      "I492.7" { ExternalVisible := 'False'} : Bool := FALSE;   // I492.7
      "I493.0" { ExternalVisible := 'False'} : Bool := FALSE;   // I493.0
      "I493.1" { ExternalVisible := 'False'} : Bool := FALSE;   // I493.1
      "I493.2" { ExternalVisible := 'False'} : Bool := FALSE;   // I493.2
      "I493.3" { ExternalVisible := 'False'} : Bool := FALSE;   // I493.3
      "I493.4" { ExternalVisible := 'False'} : Bool := FALSE;   // I493.4
      "I493.5" { ExternalVisible := 'False'} : Bool := FALSE;   // I493.5
      "I493.6" { ExternalVisible := 'False'} : Bool := FALSE;   // I493.6
      "I493.7" { ExternalVisible := 'False'} : Bool := FALSE;   // I493.7
      "I494.0" { ExternalVisible := 'False'} : Bool := FALSE;   // I494.0
      "I494.1" { ExternalVisible := 'False'} : Bool := FALSE;   // I494.1
      "I494.2" { ExternalVisible := 'False'} : Bool := FALSE;   // I494.2
      "I494.3" { ExternalVisible := 'False'} : Bool := FALSE;   // I494.3
      "I494.4" { ExternalVisible := 'False'} : Bool := FALSE;   // I494.4
      "I494.5" { ExternalVisible := 'False'} : Bool := FALSE;   // I494.5
      "I494.6" { ExternalVisible := 'False'} : Bool := FALSE;   // I494.6
      "I494.7" { ExternalVisible := 'False'} : Bool := FALSE;   // I494.7
      "I495.0" { ExternalVisible := 'False'} : Bool := FALSE;   // I495.0
      "I495.1" { ExternalVisible := 'False'} : Bool := FALSE;   // I495.1
      "I495.2" { ExternalVisible := 'False'} : Bool := FALSE;   // I495.2
      "I495.3" { ExternalVisible := 'False'} : Bool := FALSE;   // I495.3
      "I495.4" { ExternalVisible := 'False'} : Bool := FALSE;   // I495.4
      "I495.5" { ExternalVisible := 'False'} : Bool := FALSE;   // I495.5
      "I495.6" { ExternalVisible := 'False'} : Bool := FALSE;   // I495.6
      "I495.7" { ExternalVisible := 'False'} : Bool := FALSE;   // I495.7
      "I496.0" { ExternalVisible := 'False'} : Bool := FALSE;   // I496.0
      "I496.1" { ExternalVisible := 'False'} : Bool := FALSE;   // I496.1
      "I496.2" { ExternalVisible := 'False'} : Bool := FALSE;   // I496.2
      "I496.3" { ExternalVisible := 'False'} : Bool := FALSE;   // I496.3
      "I496.4" { ExternalVisible := 'False'} : Bool := FALSE;   // I496.4
      "I496.5" { ExternalVisible := 'False'} : Bool := FALSE;   // I496.5
      "I496.6" { ExternalVisible := 'False'} : Bool := FALSE;   // I496.6
      "I496.7" { ExternalVisible := 'False'} : Bool := FALSE;   // I496.7
      "I497.0" { ExternalVisible := 'False'} : Bool := FALSE;   // I497.0
      "I497.1" { ExternalVisible := 'False'} : Bool := FALSE;   // I497.1
      "I497.2" { ExternalVisible := 'False'} : Bool := FALSE;   // I497.2
      "I497.3" { ExternalVisible := 'False'} : Bool := FALSE;   // I497.3
      "I497.4" { ExternalVisible := 'False'} : Bool := FALSE;   // I497.4
      "I497.5" { ExternalVisible := 'False'} : Bool := FALSE;   // I497.5
      "I497.6" { ExternalVisible := 'False'} : Bool := FALSE;   // I497.6
      "I497.7" { ExternalVisible := 'False'} : Bool := FALSE;   // I497.7
      "I498.0" { ExternalVisible := 'False'} : Bool := FALSE;   // I498.0
      "I498.1" { ExternalVisible := 'False'} : Bool := FALSE;   // I498.1
      "I498.2" { ExternalVisible := 'False'} : Bool := FALSE;   // I498.2
      "I498.3" { ExternalVisible := 'False'} : Bool := FALSE;   // I498.3
      "I498.4" { ExternalVisible := 'False'} : Bool := FALSE;   // I498.4
      "I498.5" { ExternalVisible := 'False'} : Bool := FALSE;   // I498.5
      "I498.6" { ExternalVisible := 'False'} : Bool := FALSE;   // I498.6
      "I498.7" { ExternalVisible := 'False'} : Bool := FALSE;   // I498.7
      "I499.0" { ExternalVisible := 'False'} : Bool := FALSE;   // I499.0
      "I499.1" { ExternalVisible := 'False'} : Bool := FALSE;   // I499.1
      "I499.2" { ExternalVisible := 'False'} : Bool := FALSE;   // I499.2
      "I499.3" { ExternalVisible := 'False'} : Bool := FALSE;   // I499.3
      "I499.4" { ExternalVisible := 'False'} : Bool := FALSE;   // I499.4
      "I499.5" { ExternalVisible := 'False'} : Bool := FALSE;   // I499.5
      "I499.6" { ExternalVisible := 'False'} : Bool := FALSE;   // I499.6
      "I499.7" { ExternalVisible := 'False'} : Bool := FALSE;   // I499.7
      V01_Home { ExternalVisible := 'False'} : Bool := FALSE;   // 送料气缸缩回
      "V01-Work" { ExternalVisible := 'False'} : Bool := FALSE;   // 送料气缸伸出
      "V02-Home" { ExternalVisible := 'False'} : Bool := FALSE;   // 定子定位气缸缩回
      "V02-Work" { ExternalVisible := 'False'} : Bool := FALSE;   // 定子定位气缸伸出
      "V03-Home" { ExternalVisible := 'False'} : Bool := FALSE;   // 压紧气缸缩回
      "V03-Work" { ExternalVisible := 'False'} : Bool := FALSE;   // 压紧气缸伸出
      "V04-Home1" { ExternalVisible := 'False'} : Bool := FALSE;   // 纸切断气缸1缩回
      "V04-Work1" { ExternalVisible := 'False'} : Bool := FALSE;   // 纸切断气缸1伸出
      V05_Home1 { ExternalVisible := 'False'} : Bool := FALSE;   // 产品推出气缸1缩回
      V05_Work1 { ExternalVisible := 'False'} : Bool := FALSE;   // 产品推出气缸1伸出
      V06_Home1 { ExternalVisible := 'False'} : Bool := FALSE;   // 推纸气缸1缩回
      V06_Work1 { ExternalVisible := 'False'} : Bool := FALSE;   // 推纸气缸1伸出
      V07_Home1 { ExternalVisible := 'False'} : Bool := FALSE;   // 纸夹持气缸1缩回
      V07_Work1 { ExternalVisible := 'False'} : Bool := FALSE;   // 纸夹持气缸1伸出
      V08_Home1 { ExternalVisible := 'False'} : Bool := FALSE;   // 压纸气缸1缩回
      V08_Work1 { ExternalVisible := 'False'} : Bool := FALSE;   // 压纸气缸1伸出
      PX1 { ExternalVisible := 'False'} : Bool := FALSE;   // 左侧绝缘纸插入到位传感器
      PX2 { ExternalVisible := 'False'} : Bool := FALSE;   // 右侧绝缘纸插入到位传感器
      PX3 { ExternalVisible := 'False'} : Bool := FALSE;   // 左侧纸有无检测传感器
      PX4 { ExternalVisible := 'False'} : Bool := FALSE;   // 右侧纸有无检测传感器
      PX5 { ExternalVisible := 'False'} : Bool := FALSE;   // 左侧纸长限位1
      PX6 { ExternalVisible := 'False'} : Bool := FALSE;   // 左侧纸长限位2
      "V04-Home2" { ExternalVisible := 'False'} : Bool := FALSE;   // 纸切断气缸2缩回
      "V04-Work2" { ExternalVisible := 'False'} : Bool := FALSE;   // 纸切断气缸2伸出
      V05_Home2 { ExternalVisible := 'False'} : Bool := FALSE;   // 产品推出气缸2缩回
      V05_Work2 { ExternalVisible := 'False'} : Bool := FALSE;   // 产品推出气缸2伸出
      V06_Home2 { ExternalVisible := 'False'} : Bool := FALSE;   // 推纸气缸2缩回
      V06_Work2 { ExternalVisible := 'False'} : Bool := FALSE;   // 推纸气缸2伸出
      V07_Home2 { ExternalVisible := 'False'} : Bool := FALSE;   // 纸夹持气缸2缩回
      V07_Work2 { ExternalVisible := 'False'} : Bool := FALSE;   // 纸夹持气缸伸出
      V08_Home2 { ExternalVisible := 'False'} : Bool := FALSE;   // 压纸气缸2缩回
      V08_Work2 { ExternalVisible := 'False'} : Bool := FALSE;   // 压纸气缸2伸出
      V09_Home { ExternalVisible := 'False'} : Bool := FALSE;   // 定位开关气缸缩回
      "V09-Work" { ExternalVisible := 'False'} : Bool := FALSE;   // 定位开关气缸伸出
      PX7 { ExternalVisible := 'False'} : Bool := FALSE;   // 右侧纸长限位1
      PX8 { ExternalVisible := 'False'} : Bool := FALSE;   // 右侧纸长限位2
      "I504.4" { ExternalVisible := 'False'} : Bool := FALSE;   // 备用
      "I504.5" { ExternalVisible := 'False'} : Bool := FALSE;   // 备用
      "I504.6" { ExternalVisible := 'False'} : Bool := FALSE;   // 备用
      "I504.7" { ExternalVisible := 'False'} : Bool := FALSE;   // 备用
      "I505.0" { ExternalVisible := 'False'} : Bool := FALSE;   // 备用
      "I505.1" { ExternalVisible := 'False'} : Bool := FALSE;   // 备用
      "I505.2" { ExternalVisible := 'False'} : Bool := FALSE;   // 备用
      "I505.3" { ExternalVisible := 'False'} : Bool := FALSE;   // 备用
      "I505.4" { ExternalVisible := 'False'} : Bool := FALSE;   // 备用
      "I505.5" { ExternalVisible := 'False'} : Bool := FALSE;   // 备用
      "I505.6" { ExternalVisible := 'False'} : Bool := FALSE;   // 备用
      "I505.7" { ExternalVisible := 'False'} : Bool := FALSE;   // 备用
      "I506.0" { ExternalVisible := 'False'} : Bool := FALSE;   // I506.0
      "I506.1" { ExternalVisible := 'False'} : Bool := FALSE;   // I506.1
      "I506.2" { ExternalVisible := 'False'} : Bool := FALSE;   // I506.2
      "I506.3" { ExternalVisible := 'False'} : Bool := FALSE;   // I506.3
      "I506.4" { ExternalVisible := 'False'} : Bool := FALSE;   // I506.4
      "I506.5" { ExternalVisible := 'False'} : Bool := FALSE;   // I506.5
      "I506.6" { ExternalVisible := 'False'} : Bool := FALSE;   // I506.6
      "I506.7" { ExternalVisible := 'False'} : Bool := FALSE;   // I506.7
      "I507.0" { ExternalVisible := 'False'} : Bool := FALSE;   // I507.0
      "I507.1" { ExternalVisible := 'False'} : Bool := FALSE;   // I507.1
      "I507.2" { ExternalVisible := 'False'} : Bool := FALSE;   // I507.2
      "I507.3" { ExternalVisible := 'False'} : Bool := FALSE;   // I507.3
      "I507.4" { ExternalVisible := 'False'} : Bool := FALSE;   // I507.4
      "I507.5" { ExternalVisible := 'False'} : Bool := FALSE;   // I507.5
      "I507.6" { ExternalVisible := 'False'} : Bool := FALSE;   // I507.6
      "I507.7" { ExternalVisible := 'False'} : Bool := FALSE;   // I507.7
      "I508.0" { ExternalVisible := 'False'} : Bool := FALSE;   // I508.0
      "I508.1" { ExternalVisible := 'False'} : Bool := FALSE;   // I508.1
      "I508.2" { ExternalVisible := 'False'} : Bool := FALSE;   // I508.2
      "I508.3" { ExternalVisible := 'False'} : Bool := FALSE;   // I508.3
      "I508.4" { ExternalVisible := 'False'} : Bool := FALSE;   // I508.4
      "I508.5" { ExternalVisible := 'False'} : Bool := FALSE;   // I508.5
      "I508.6" { ExternalVisible := 'False'} : Bool := FALSE;   // I508.6
      "I508.7" { ExternalVisible := 'False'} : Bool := FALSE;   // I508.7
      "I509.0" { ExternalVisible := 'False'} : Bool := FALSE;   // I509.0
      "I509.1" { ExternalVisible := 'False'} : Bool := FALSE;   // I509.1
      "I509.2" { ExternalVisible := 'False'} : Bool := FALSE;   // I509.2
      "I509.3" { ExternalVisible := 'False'} : Bool := FALSE;   // I509.3
      "I509.4" { ExternalVisible := 'False'} : Bool := FALSE;   // I509.4
      "I509.5" { ExternalVisible := 'False'} : Bool := FALSE;   // I509.5
      "I509.6" { ExternalVisible := 'False'} : Bool := FALSE;   // I509.6
      "I509.7" { ExternalVisible := 'False'} : Bool := FALSE;   // I509.7
      "I510.0" { ExternalVisible := 'False'} : Bool := FALSE;   // I510.0
      "I510.1" { ExternalVisible := 'False'} : Bool := FALSE;   // I510.1
      "I510.2" { ExternalVisible := 'False'} : Bool := FALSE;   // I510.2
      "I510.3" { ExternalVisible := 'False'} : Bool := FALSE;   // I510.3
      "I510.4" { ExternalVisible := 'False'} : Bool := FALSE;   // I510.4
      "I510.5" { ExternalVisible := 'False'} : Bool := FALSE;   // I510.5
      "I510.6" { ExternalVisible := 'False'} : Bool := FALSE;   // I510.6
      "I510.7" { ExternalVisible := 'False'} : Bool := FALSE;   // I510.7
      "I511.0" { ExternalVisible := 'False'} : Bool := FALSE;   // I511.0
      "I511.1" { ExternalVisible := 'False'} : Bool := FALSE;   // I511.1
      "I511.2" { ExternalVisible := 'False'} : Bool := FALSE;   // I511.2
      "I511.3" { ExternalVisible := 'False'} : Bool := FALSE;   // I511.3
      "I511.4" { ExternalVisible := 'False'} : Bool := FALSE;   // I511.4
      "I511.5" { ExternalVisible := 'False'} : Bool := FALSE;   // I511.5
      "I511.6" { ExternalVisible := 'False'} : Bool := FALSE;   // I511.6
      "I511.7" { ExternalVisible := 'False'} : Bool := FALSE;   // I511.7
      "I512.0" { ExternalVisible := 'False'} : Bool := FALSE;   // I512.0
      "I512.1" { ExternalVisible := 'False'} : Bool := FALSE;   // I512.1
      "I512.2" { ExternalVisible := 'False'} : Bool := FALSE;   // I512.2
      "I512.3" { ExternalVisible := 'False'} : Bool := FALSE;   // I512.3
      "I512.4" { ExternalVisible := 'False'} : Bool := FALSE;   // I512.4
      "I512.5" { ExternalVisible := 'False'} : Bool := FALSE;   // I512.5
      "I512.6" { ExternalVisible := 'False'} : Bool := FALSE;   // I512.6
      "I512.7" { ExternalVisible := 'False'} : Bool := FALSE;   // I512.7
      "I513.0" { ExternalVisible := 'False'} : Bool := FALSE;   // I513.0
      "I513.1" { ExternalVisible := 'False'} : Bool := FALSE;   // I513.1
      "I513.2" { ExternalVisible := 'False'} : Bool := FALSE;   // I513.2
      "I513.3" { ExternalVisible := 'False'} : Bool := FALSE;   // I513.3
      "I513.4" { ExternalVisible := 'False'} : Bool := FALSE;   // I513.4
      "I513.5" { ExternalVisible := 'False'} : Bool := FALSE;   // I513.5
      "I513.6" { ExternalVisible := 'False'} : Bool := FALSE;   // I513.6
      "I513.7" { ExternalVisible := 'False'} : Bool := FALSE;   // I513.7
      "I514.0" { ExternalVisible := 'False'} : Bool := FALSE;   // I514.0
      "I514.1" { ExternalVisible := 'False'} : Bool := FALSE;   // I514.1
      "I514.2" { ExternalVisible := 'False'} : Bool := FALSE;   // I514.2
      "I514.3" { ExternalVisible := 'False'} : Bool := FALSE;   // I514.3
      "I514.4" { ExternalVisible := 'False'} : Bool := FALSE;   // I514.4
      "I514.5" { ExternalVisible := 'False'} : Bool := FALSE;   // I514.5
      "I514.6" { ExternalVisible := 'False'} : Bool := FALSE;   // I514.6
      "I514.7" { ExternalVisible := 'False'} : Bool := FALSE;   // I514.7
      "I515.0" { ExternalVisible := 'False'} : Bool := FALSE;   // I515.0
      "I515.1" { ExternalVisible := 'False'} : Bool := FALSE;   // I515.1
      "I515.2" { ExternalVisible := 'False'} : Bool := FALSE;   // I515.2
      "I515.3" { ExternalVisible := 'False'} : Bool := FALSE;   // I515.3
      "I515.4" { ExternalVisible := 'False'} : Bool := FALSE;   // I515.4
      "I515.5" { ExternalVisible := 'False'} : Bool := FALSE;   // I515.5
      "I515.6" { ExternalVisible := 'False'} : Bool := FALSE;   // I515.6
      "I515.7" { ExternalVisible := 'False'} : Bool := FALSE;   // I515.7
      "I516.0" { ExternalVisible := 'False'} : Bool := FALSE;   // I516.0
      "I516.1" { ExternalVisible := 'False'} : Bool := FALSE;   // I516.1
      "I516.2" { ExternalVisible := 'False'} : Bool := FALSE;   // I516.2
      "I516.3" { ExternalVisible := 'False'} : Bool := FALSE;   // I516.3
      "I516.4" { ExternalVisible := 'False'} : Bool := FALSE;   // I516.4
      "I516.5" { ExternalVisible := 'False'} : Bool := FALSE;   // I516.5
      "I516.6" { ExternalVisible := 'False'} : Bool := FALSE;   // I516.6
      "I516.7" { ExternalVisible := 'False'} : Bool := FALSE;   // I516.7
      "I517.0" { ExternalVisible := 'False'} : Bool := FALSE;   // I517.0
      "I517.1" { ExternalVisible := 'False'} : Bool := FALSE;   // I517.1
      "I517.2" { ExternalVisible := 'False'} : Bool := FALSE;   // I517.2
      "I517.3" { ExternalVisible := 'False'} : Bool := FALSE;   // I517.3
      "I517.4" { ExternalVisible := 'False'} : Bool := FALSE;   // I517.4
      "I517.5" { ExternalVisible := 'False'} : Bool := FALSE;   // I517.5
      "I517.6" { ExternalVisible := 'False'} : Bool := FALSE;   // I517.6
      "I517.7" { ExternalVisible := 'False'} : Bool := FALSE;   // I517.7
      "I518.0" { ExternalVisible := 'False'} : Bool := FALSE;   // I518.0
      "I518.1" { ExternalVisible := 'False'} : Bool := FALSE;   // I518.1
      "I518.2" { ExternalVisible := 'False'} : Bool := FALSE;   // I518.2
      "I518.3" { ExternalVisible := 'False'} : Bool := FALSE;   // I518.3
      "I518.4" { ExternalVisible := 'False'} : Bool := FALSE;   // I518.4
      "I518.5" { ExternalVisible := 'False'} : Bool := FALSE;   // I518.5
      "I518.6" { ExternalVisible := 'False'} : Bool := FALSE;   // I518.6
      "I518.7" { ExternalVisible := 'False'} : Bool := FALSE;   // I518.7
      "I519.0" { ExternalVisible := 'False'} : Bool := FALSE;   // I519.0
      "I519.1" { ExternalVisible := 'False'} : Bool := FALSE;   // I519.1
      "I519.2" { ExternalVisible := 'False'} : Bool := FALSE;   // I519.2
      "I519.3" { ExternalVisible := 'False'} : Bool := FALSE;   // I519.3
      "I519.4" { ExternalVisible := 'False'} : Bool := FALSE;   // I519.4
      "I519.5" { ExternalVisible := 'False'} : Bool := FALSE;   // I519.5
      "I519.6" { ExternalVisible := 'False'} : Bool := FALSE;   // I519.6
      "I519.7" { ExternalVisible := 'False'} : Bool := FALSE;   // I519.7
      "I520.0" { ExternalVisible := 'False'} : Bool := FALSE;   // I520.0
      "I520.1" { ExternalVisible := 'False'} : Bool := FALSE;   // I520.1
      "I520.2" { ExternalVisible := 'False'} : Bool := FALSE;   // I520.2
      "I520.3" { ExternalVisible := 'False'} : Bool := FALSE;   // I520.3
      "I520.4" { ExternalVisible := 'False'} : Bool := FALSE;   // I520.4
      "I520.5" { ExternalVisible := 'False'} : Bool := FALSE;   // I520.5
      "I520.6" { ExternalVisible := 'False'} : Bool := FALSE;   // I520.6
      "I520.7" { ExternalVisible := 'False'} : Bool := FALSE;   // I520.7
      "I521.0" { ExternalVisible := 'False'} : Bool := FALSE;   // I521.0
      "I521.1" { ExternalVisible := 'False'} : Bool := FALSE;   // I521.1
      "I521.2" { ExternalVisible := 'False'} : Bool := FALSE;   // I521.2
      "I521.3" { ExternalVisible := 'False'} : Bool := FALSE;   // I521.3
      "I521.4" { ExternalVisible := 'False'} : Bool := FALSE;   // I521.4
      "I521.5" { ExternalVisible := 'False'} : Bool := FALSE;   // I521.5
      "I521.6" { ExternalVisible := 'False'} : Bool := FALSE;   // I521.6
      "I521.7" { ExternalVisible := 'False'} : Bool := FALSE;   // I521.7
      "I522.0" { ExternalVisible := 'False'} : Bool := FALSE;   // I522.0
      "I522.1" { ExternalVisible := 'False'} : Bool := FALSE;   // I522.1
      "I522.2" { ExternalVisible := 'False'} : Bool := FALSE;   // I522.2
      "I522.3" { ExternalVisible := 'False'} : Bool := FALSE;   // I522.3
      "I522.4" { ExternalVisible := 'False'} : Bool := FALSE;   // I522.4
      "I522.5" { ExternalVisible := 'False'} : Bool := FALSE;   // I522.5
      "I522.6" { ExternalVisible := 'False'} : Bool := FALSE;   // I522.6
      "I522.7" { ExternalVisible := 'False'} : Bool := FALSE;   // I522.7
      "I523.0" { ExternalVisible := 'False'} : Bool := FALSE;   // I523.0
      "I523.1" { ExternalVisible := 'False'} : Bool := FALSE;   // I523.1
      "I523.2" { ExternalVisible := 'False'} : Bool := FALSE;   // I523.2
      "I523.3" { ExternalVisible := 'False'} : Bool := FALSE;   // I523.3
      "I523.4" { ExternalVisible := 'False'} : Bool := FALSE;   // I523.4
      "I523.5" { ExternalVisible := 'False'} : Bool := FALSE;   // I523.5
      "I523.6" { ExternalVisible := 'False'} : Bool := FALSE;   // I523.6
      "I523.7" { ExternalVisible := 'False'} : Bool := FALSE;   // I523.7
      "I524.0" { ExternalVisible := 'False'} : Bool := FALSE;   // I524.0
      "I524.1" { ExternalVisible := 'False'} : Bool := FALSE;   // I524.1
      "I524.2" { ExternalVisible := 'False'} : Bool := FALSE;   // I524.2
      "I524.3" { ExternalVisible := 'False'} : Bool := FALSE;   // I524.3
      "I524.4" { ExternalVisible := 'False'} : Bool := FALSE;   // I524.4
      "I524.5" { ExternalVisible := 'False'} : Bool := FALSE;   // I524.5
      "I524.6" { ExternalVisible := 'False'} : Bool := FALSE;   // I524.6
      "I524.7" { ExternalVisible := 'False'} : Bool := FALSE;   // I524.7
      "I525.0" { ExternalVisible := 'False'} : Bool := FALSE;   // I525.0
      "I525.1" { ExternalVisible := 'False'} : Bool := FALSE;   // I525.1
      "I525.2" { ExternalVisible := 'False'} : Bool := FALSE;   // I525.2
      "I525.3" { ExternalVisible := 'False'} : Bool := FALSE;   // I525.3
      "I525.4" { ExternalVisible := 'False'} : Bool := FALSE;   // I525.4
      "I525.5" { ExternalVisible := 'False'} : Bool := FALSE;   // I525.5
      "I525.6" { ExternalVisible := 'False'} : Bool := FALSE;   // I525.6
      "I525.7" { ExternalVisible := 'False'} : Bool := FALSE;   // I525.7
      "I526.0" { ExternalVisible := 'False'} : Bool := FALSE;   // I526.0
      "I526.1" { ExternalVisible := 'False'} : Bool := FALSE;   // I526.1
      "I526.2" { ExternalVisible := 'False'} : Bool := FALSE;   // I526.2
      "I526.3" { ExternalVisible := 'False'} : Bool := FALSE;   // I526.3
      "I526.4" { ExternalVisible := 'False'} : Bool := FALSE;   // I526.4
      "I526.5" { ExternalVisible := 'False'} : Bool := FALSE;   // I526.5
      "I526.6" { ExternalVisible := 'False'} : Bool := FALSE;   // I526.6
      "I526.7" { ExternalVisible := 'False'} : Bool := FALSE;   // I526.7
      "I527.0" { ExternalVisible := 'False'} : Bool := FALSE;   // I527.0
      "I527.1" { ExternalVisible := 'False'} : Bool := FALSE;   // I527.1
      "I527.2" { ExternalVisible := 'False'} : Bool := FALSE;   // I527.2
      "I527.3" { ExternalVisible := 'False'} : Bool := FALSE;   // I527.3
      "I527.4" { ExternalVisible := 'False'} : Bool := FALSE;   // I527.4
      "I527.5" { ExternalVisible := 'False'} : Bool := FALSE;   // I527.5
      "I527.6" { ExternalVisible := 'False'} : Bool := FALSE;   // I527.6
      "I527.7" { ExternalVisible := 'False'} : Bool := FALSE;   // I527.7
      "I528.0" { ExternalVisible := 'False'} : Bool := FALSE;   // I528.0
      "I528.1" { ExternalVisible := 'False'} : Bool := FALSE;   // I528.1
      "I528.2" { ExternalVisible := 'False'} : Bool := FALSE;   // I528.2
      "I528.3" { ExternalVisible := 'False'} : Bool := FALSE;   // I528.3
      "I528.4" { ExternalVisible := 'False'} : Bool := FALSE;   // I528.4
      "I528.5" { ExternalVisible := 'False'} : Bool := FALSE;   // I528.5
      "I528.6" { ExternalVisible := 'False'} : Bool := FALSE;   // I528.6
      "I528.7" { ExternalVisible := 'False'} : Bool := FALSE;   // I528.7
      "I529.0" { ExternalVisible := 'False'} : Bool := FALSE;   // I529.0
      "I529.1" { ExternalVisible := 'False'} : Bool := FALSE;   // I529.1
      "I529.2" { ExternalVisible := 'False'} : Bool := FALSE;   // I529.2
      "I529.3" { ExternalVisible := 'False'} : Bool := FALSE;   // I529.3
      "I529.4" { ExternalVisible := 'False'} : Bool := FALSE;   // I529.4
      "I529.5" { ExternalVisible := 'False'} : Bool := FALSE;   // I529.5
      "I529.6" { ExternalVisible := 'False'} : Bool := FALSE;   // I529.6
      "I529.7" { ExternalVisible := 'False'} : Bool := FALSE;   // I529.7
      "I530.0" { ExternalVisible := 'False'} : Bool := FALSE;   // I530.0
      "I530.1" { ExternalVisible := 'False'} : Bool := FALSE;   // I530.1
      "I530.2" { ExternalVisible := 'False'} : Bool := FALSE;   // I530.2
      "I530.3" { ExternalVisible := 'False'} : Bool := FALSE;   // I530.3
      "I530.4" { ExternalVisible := 'False'} : Bool := FALSE;   // I530.4
      "I530.5" { ExternalVisible := 'False'} : Bool := FALSE;   // I530.5
      "I530.6" { ExternalVisible := 'False'} : Bool := FALSE;   // I530.6
      "I530.7" { ExternalVisible := 'False'} : Bool := FALSE;   // I530.7
      "I531.0" { ExternalVisible := 'False'} : Bool := FALSE;   // I531.0
      "I531.1" { ExternalVisible := 'False'} : Bool := FALSE;   // I531.1
      "I531.2" { ExternalVisible := 'False'} : Bool := FALSE;   // I531.2
      "I531.3" { ExternalVisible := 'False'} : Bool := FALSE;   // I531.3
      "I531.4" { ExternalVisible := 'False'} : Bool := FALSE;   // I531.4
      "I531.5" { ExternalVisible := 'False'} : Bool := FALSE;   // I531.5
      "I531.6" { ExternalVisible := 'False'} : Bool := FALSE;   // I531.6
      "I531.7" { ExternalVisible := 'False'} : Bool := FALSE;   // I531.7
      "I532.0" { ExternalVisible := 'False'} : Bool := FALSE;   // I532.0
      "I532.1" { ExternalVisible := 'False'} : Bool := FALSE;   // I532.1
      "I532.2" { ExternalVisible := 'False'} : Bool := FALSE;   // I532.2
      "I532.3" { ExternalVisible := 'False'} : Bool := FALSE;   // I532.3
      "I532.4" { ExternalVisible := 'False'} : Bool := FALSE;   // I532.4
      "I532.5" { ExternalVisible := 'False'} : Bool := FALSE;   // I532.5
      "I532.6" { ExternalVisible := 'False'} : Bool := FALSE;   // I532.6
      "I532.7" { ExternalVisible := 'False'} : Bool := FALSE;   // I532.7
      "I533.0" { ExternalVisible := 'False'} : Bool := FALSE;   // I533.0
      "I533.1" { ExternalVisible := 'False'} : Bool := FALSE;   // I533.1
      "I533.2" { ExternalVisible := 'False'} : Bool := FALSE;   // I533.2
      "I533.3" { ExternalVisible := 'False'} : Bool := FALSE;   // I533.3
      "I533.4" { ExternalVisible := 'False'} : Bool := FALSE;   // I533.4
      "I533.5" { ExternalVisible := 'False'} : Bool := FALSE;   // I533.5
      "I533.6" { ExternalVisible := 'False'} : Bool := FALSE;   // I533.6
      "I533.7" { ExternalVisible := 'False'} : Bool := FALSE;   // I533.7
      "I534.0" { ExternalVisible := 'False'} : Bool := FALSE;   // I534.0
      "I534.1" { ExternalVisible := 'False'} : Bool := FALSE;   // I534.1
      "I534.2" { ExternalVisible := 'False'} : Bool := FALSE;   // I534.2
      "I534.3" { ExternalVisible := 'False'} : Bool := FALSE;   // I534.3
      "I534.4" { ExternalVisible := 'False'} : Bool := FALSE;   // I534.4
      "I534.5" { ExternalVisible := 'False'} : Bool := FALSE;   // I534.5
      "I534.6" { ExternalVisible := 'False'} : Bool := FALSE;   // I534.6
      "I534.7" { ExternalVisible := 'False'} : Bool := FALSE;   // I534.7
      "I535.0" { ExternalVisible := 'False'} : Bool := FALSE;   // I535.0
      "I535.1" { ExternalVisible := 'False'} : Bool := FALSE;   // I535.1
      "I535.2" { ExternalVisible := 'False'} : Bool := FALSE;   // I535.2
      "I535.3" { ExternalVisible := 'False'} : Bool := FALSE;   // I535.3
      "I535.4" { ExternalVisible := 'False'} : Bool := FALSE;   // I535.4
      "I535.5" { ExternalVisible := 'False'} : Bool := FALSE;   // I535.5
      "I535.6" { ExternalVisible := 'False'} : Bool := FALSE;   // I535.6
      "I535.7" { ExternalVisible := 'False'} : Bool := FALSE;   // I535.7
      "I536.0" { ExternalVisible := 'False'} : Bool := FALSE;   // I536.0
      "I536.1" { ExternalVisible := 'False'} : Bool := FALSE;   // I536.1
      "I536.2" { ExternalVisible := 'False'} : Bool := FALSE;   // I536.2
      "I536.3" { ExternalVisible := 'False'} : Bool := FALSE;   // I536.3
      "I536.4" { ExternalVisible := 'False'} : Bool := FALSE;   // I536.4
      "I536.5" { ExternalVisible := 'False'} : Bool := FALSE;   // I536.5
      "I536.6" { ExternalVisible := 'False'} : Bool := FALSE;   // I536.6
      "I536.7" { ExternalVisible := 'False'} : Bool := FALSE;   // I536.7
      "I537.0" { ExternalVisible := 'False'} : Bool := FALSE;   // I537.0
      "I537.1" { ExternalVisible := 'False'} : Bool := FALSE;   // I537.1
      "I537.2" { ExternalVisible := 'False'} : Bool := FALSE;   // I537.2
      "I537.3" { ExternalVisible := 'False'} : Bool := FALSE;   // I537.3
      "I537.4" { ExternalVisible := 'False'} : Bool := FALSE;   // I537.4
      "I537.5" { ExternalVisible := 'False'} : Bool := FALSE;   // I537.5
      "I537.6" { ExternalVisible := 'False'} : Bool := FALSE;   // I537.6
      "I537.7" { ExternalVisible := 'False'} : Bool := FALSE;   // I537.7
      "I538.0" { ExternalVisible := 'False'} : Bool := FALSE;   // I538.0
      "I538.1" { ExternalVisible := 'False'} : Bool := FALSE;   // I538.1
      "I538.2" { ExternalVisible := 'False'} : Bool := FALSE;   // I538.2
      "I538.3" { ExternalVisible := 'False'} : Bool := FALSE;   // I538.3
      "I538.4" { ExternalVisible := 'False'} : Bool := FALSE;   // I538.4
      "I538.5" { ExternalVisible := 'False'} : Bool := FALSE;   // I538.5
      "I538.6" { ExternalVisible := 'False'} : Bool := FALSE;   // I538.6
      "I538.7" { ExternalVisible := 'False'} : Bool := FALSE;   // I538.7
      "I539.0" { ExternalVisible := 'False'} : Bool := FALSE;   // I539.0
      "I539.1" { ExternalVisible := 'False'} : Bool := FALSE;   // I539.1
      "I539.2" { ExternalVisible := 'False'} : Bool := FALSE;   // I539.2
      "I539.3" { ExternalVisible := 'False'} : Bool := FALSE;   // I539.3
      "I539.4" { ExternalVisible := 'False'} : Bool := FALSE;   // I539.4
      "I539.5" { ExternalVisible := 'False'} : Bool := FALSE;   // I539.5
      "I539.6" { ExternalVisible := 'False'} : Bool := FALSE;   // I539.6
      "I539.7" { ExternalVisible := 'False'} : Bool := FALSE;   // I539.7
      "I540.0" { ExternalVisible := 'False'} : Bool := FALSE;   // I540.0
      "I540.1" { ExternalVisible := 'False'} : Bool := FALSE;   // I540.1
      "I540.2" { ExternalVisible := 'False'} : Bool := FALSE;   // I540.2
      "I540.3" { ExternalVisible := 'False'} : Bool := FALSE;   // I540.3
      "I540.4" { ExternalVisible := 'False'} : Bool := FALSE;   // I540.4
      "I540.5" { ExternalVisible := 'False'} : Bool := FALSE;   // I540.5
      "I540.6" { ExternalVisible := 'False'} : Bool := FALSE;   // I540.6
      "I540.7" { ExternalVisible := 'False'} : Bool := FALSE;   // I540.7
      "I541.0" { ExternalVisible := 'False'} : Bool := FALSE;   // I541.0
      "I541.1" { ExternalVisible := 'False'} : Bool := FALSE;   // I541.1
      "I541.2" { ExternalVisible := 'False'} : Bool := FALSE;   // I541.2
      "I541.3" { ExternalVisible := 'False'} : Bool := FALSE;   // I541.3
      "I541.4" { ExternalVisible := 'False'} : Bool := FALSE;   // I541.4
      "I541.5" { ExternalVisible := 'False'} : Bool := FALSE;   // I541.5
      "I541.6" { ExternalVisible := 'False'} : Bool := FALSE;   // I541.6
      "I541.7" { ExternalVisible := 'False'} : Bool := FALSE;   // I541.7
      "I542.0" { ExternalVisible := 'False'} : Bool := FALSE;   // I542.0
      "I542.1" { ExternalVisible := 'False'} : Bool := FALSE;   // I542.1
      "I542.2" { ExternalVisible := 'False'} : Bool := FALSE;   // I542.2
      "I542.3" { ExternalVisible := 'False'} : Bool := FALSE;   // I542.3
      "I542.4" { ExternalVisible := 'False'} : Bool := FALSE;   // I542.4
      "I542.5" { ExternalVisible := 'False'} : Bool := FALSE;   // I542.5
      "I542.6" { ExternalVisible := 'False'} : Bool := FALSE;   // I542.6
      "I542.7" { ExternalVisible := 'False'} : Bool := FALSE;   // I542.7
      "I543.0" { ExternalVisible := 'False'} : Bool := FALSE;   // I543.0
      "I543.1" { ExternalVisible := 'False'} : Bool := FALSE;   // I543.1
      "I543.2" { ExternalVisible := 'False'} : Bool := FALSE;   // I543.2
      "I543.3" { ExternalVisible := 'False'} : Bool := FALSE;   // I543.3
      "I543.4" { ExternalVisible := 'False'} : Bool := FALSE;   // I543.4
      "I543.5" { ExternalVisible := 'False'} : Bool := FALSE;   // I543.5
      "I543.6" { ExternalVisible := 'False'} : Bool := FALSE;   // I543.6
      "I543.7" { ExternalVisible := 'False'} : Bool := FALSE;   // I543.7
      "I544.0" { ExternalVisible := 'False'} : Bool := FALSE;   // I544.0
      "I544.1" { ExternalVisible := 'False'} : Bool := FALSE;   // I544.1
      "I544.2" { ExternalVisible := 'False'} : Bool := FALSE;   // I544.2
      "I544.3" { ExternalVisible := 'False'} : Bool := FALSE;   // I544.3
      "I544.4" { ExternalVisible := 'False'} : Bool := FALSE;   // I544.4
      "I544.5" { ExternalVisible := 'False'} : Bool := FALSE;   // I544.5
      "I544.6" { ExternalVisible := 'False'} : Bool := FALSE;   // I544.6
      "I544.7" { ExternalVisible := 'False'} : Bool := FALSE;   // I544.7
      "I545.0" { ExternalVisible := 'False'} : Bool := FALSE;   // I545.0
      "I545.1" { ExternalVisible := 'False'} : Bool := FALSE;   // I545.1
      "I545.2" { ExternalVisible := 'False'} : Bool := FALSE;   // I545.2
      "I545.3" { ExternalVisible := 'False'} : Bool := FALSE;   // I545.3
      "I545.4" { ExternalVisible := 'False'} : Bool := FALSE;   // I545.4
      "I545.5" { ExternalVisible := 'False'} : Bool := FALSE;   // I545.5
      "I545.6" { ExternalVisible := 'False'} : Bool := FALSE;   // I545.6
      "I545.7" { ExternalVisible := 'False'} : Bool := FALSE;   // I545.7
      "I546.0" { ExternalVisible := 'False'} : Bool := FALSE;   // I546.0
      "I546.1" { ExternalVisible := 'False'} : Bool := FALSE;   // I546.1
      "I546.2" { ExternalVisible := 'False'} : Bool := FALSE;   // I546.2
      "I546.3" { ExternalVisible := 'False'} : Bool := FALSE;   // I546.3
      "I546.4" { ExternalVisible := 'False'} : Bool := FALSE;   // I546.4
      "I546.5" { ExternalVisible := 'False'} : Bool := FALSE;   // I546.5
      "I546.6" { ExternalVisible := 'False'} : Bool := FALSE;   // I546.6
      "I546.7" { ExternalVisible := 'False'} : Bool := FALSE;   // I546.7
      "I547.0" { ExternalVisible := 'False'} : Bool := FALSE;   // I547.0
      "I547.1" { ExternalVisible := 'False'} : Bool := FALSE;   // I547.1
      "I547.2" { ExternalVisible := 'False'} : Bool := FALSE;   // I547.2
      "I547.3" { ExternalVisible := 'False'} : Bool := FALSE;   // I547.3
      "I547.4" { ExternalVisible := 'False'} : Bool := FALSE;   // I547.4
      "I547.5" { ExternalVisible := 'False'} : Bool := FALSE;   // I547.5
      "I547.6" { ExternalVisible := 'False'} : Bool := FALSE;   // I547.6
      "I547.7" { ExternalVisible := 'False'} : Bool := FALSE;   // I547.7
      "I548.0" { ExternalVisible := 'False'} : Bool := FALSE;   // I548.0
      "I548.1" { ExternalVisible := 'False'} : Bool := FALSE;   // I548.1
      "I548.2" { ExternalVisible := 'False'} : Bool := FALSE;   // I548.2
      "I548.3" { ExternalVisible := 'False'} : Bool := FALSE;   // I548.3
      "I548.4" { ExternalVisible := 'False'} : Bool := FALSE;   // I548.4
      "I548.5" { ExternalVisible := 'False'} : Bool := FALSE;   // I548.5
      "I548.6" { ExternalVisible := 'False'} : Bool := FALSE;   // I548.6
      "I548.7" { ExternalVisible := 'False'} : Bool := FALSE;   // I548.7
      "I549.0" { ExternalVisible := 'False'} : Bool := FALSE;   // I549.0
      "I549.1" { ExternalVisible := 'False'} : Bool := FALSE;   // I549.1
      "I549.2" { ExternalVisible := 'False'} : Bool := FALSE;   // I549.2
      "I549.3" { ExternalVisible := 'False'} : Bool := FALSE;   // I549.3
      "I549.4" { ExternalVisible := 'False'} : Bool := FALSE;   // I549.4
      "I549.5" { ExternalVisible := 'False'} : Bool := FALSE;   // I549.5
      "I549.6" { ExternalVisible := 'False'} : Bool := FALSE;   // I549.6
      "I549.7" { ExternalVisible := 'False'} : Bool := FALSE;   // I549.7
      "I550.0" { ExternalVisible := 'False'} : Bool := FALSE;   // I550.0
      "I550.1" { ExternalVisible := 'False'} : Bool := FALSE;   // I550.1
      "I550.2" { ExternalVisible := 'False'} : Bool := FALSE;   // I550.2
      "I550.3" { ExternalVisible := 'False'} : Bool := FALSE;   // I550.3
      "I550.4" { ExternalVisible := 'False'} : Bool := FALSE;   // I550.4
      "I550.5" { ExternalVisible := 'False'} : Bool := FALSE;   // I550.5
      "I550.6" { ExternalVisible := 'False'} : Bool := FALSE;   // I550.6
      "I550.7" { ExternalVisible := 'False'} : Bool := FALSE;   // I550.7
      "I551.0" { ExternalVisible := 'False'} : Bool := FALSE;   // I551.0
      "I551.1" { ExternalVisible := 'False'} : Bool := FALSE;   // I551.1
      "I551.2" { ExternalVisible := 'False'} : Bool := FALSE;   // I551.2
      "I551.3" { ExternalVisible := 'False'} : Bool := FALSE;   // I551.3
      "I551.4" { ExternalVisible := 'False'} : Bool := FALSE;   // I551.4
      "I551.5" { ExternalVisible := 'False'} : Bool := FALSE;   // I551.5
      "I551.6" { ExternalVisible := 'False'} : Bool := FALSE;   // I551.6
      "I551.7" { ExternalVisible := 'False'} : Bool := FALSE;   // I551.7
      "I552.0" { ExternalVisible := 'False'} : Bool := FALSE;   // I552.0
      "I552.1" { ExternalVisible := 'False'} : Bool := FALSE;   // I552.1
      "I552.2" { ExternalVisible := 'False'} : Bool := FALSE;   // I552.2
      "I552.3" { ExternalVisible := 'False'} : Bool := FALSE;   // I552.3
      "I552.4" { ExternalVisible := 'False'} : Bool := FALSE;   // I552.4
      "I552.5" { ExternalVisible := 'False'} : Bool := FALSE;   // I552.5
      "I552.6" { ExternalVisible := 'False'} : Bool := FALSE;   // I552.6
      "I552.7" { ExternalVisible := 'False'} : Bool := FALSE;   // I552.7
      "I553.0" { ExternalVisible := 'False'} : Bool := FALSE;   // I553.0
      "I553.1" { ExternalVisible := 'False'} : Bool := FALSE;   // I553.1
      "I553.2" { ExternalVisible := 'False'} : Bool := FALSE;   // I553.2
      "I553.3" { ExternalVisible := 'False'} : Bool := FALSE;   // I553.3
      "I553.4" { ExternalVisible := 'False'} : Bool := FALSE;   // I553.4
      "I553.5" { ExternalVisible := 'False'} : Bool := FALSE;   // I553.5
      "I553.6" { ExternalVisible := 'False'} : Bool := FALSE;   // I553.6
      "I553.7" { ExternalVisible := 'False'} : Bool := FALSE;   // I553.7
      "I554.0" { ExternalVisible := 'False'} : Bool := FALSE;   // I554.0
      "I554.1" { ExternalVisible := 'False'} : Bool := FALSE;   // I554.1
      "I554.2" { ExternalVisible := 'False'} : Bool := FALSE;   // I554.2
      "I554.3" { ExternalVisible := 'False'} : Bool := FALSE;   // I554.3
      "I554.4" { ExternalVisible := 'False'} : Bool := FALSE;   // I554.4
      "I554.5" { ExternalVisible := 'False'} : Bool := FALSE;   // I554.5
      "I554.6" { ExternalVisible := 'False'} : Bool := FALSE;   // I554.6
      "I554.7" { ExternalVisible := 'False'} : Bool := FALSE;   // I554.7
      "I555.0" { ExternalVisible := 'False'} : Bool := FALSE;   // I555.0
      "I555.1" { ExternalVisible := 'False'} : Bool := FALSE;   // I555.1
      "I555.2" { ExternalVisible := 'False'} : Bool := FALSE;   // I555.2
      "I555.3" { ExternalVisible := 'False'} : Bool := FALSE;   // I555.3
      "I555.4" { ExternalVisible := 'False'} : Bool := FALSE;   // I555.4
      "I555.5" { ExternalVisible := 'False'} : Bool := FALSE;   // I555.5
      "I555.6" { ExternalVisible := 'False'} : Bool := FALSE;   // I555.6
      "I555.7" { ExternalVisible := 'False'} : Bool := FALSE;   // I555.7
      "I556.0" { ExternalVisible := 'False'} : Bool := FALSE;   // I556.0
      "I556.1" { ExternalVisible := 'False'} : Bool := FALSE;   // I556.1
      "I556.2" { ExternalVisible := 'False'} : Bool := FALSE;   // I556.2
      "I556.3" { ExternalVisible := 'False'} : Bool := FALSE;   // I556.3
      "I556.4" { ExternalVisible := 'False'} : Bool := FALSE;   // I556.4
      "I556.5" { ExternalVisible := 'False'} : Bool := FALSE;   // I556.5
      "I556.6" { ExternalVisible := 'False'} : Bool := FALSE;   // I556.6
      "I556.7" { ExternalVisible := 'False'} : Bool := FALSE;   // I556.7
      "I557.0" { ExternalVisible := 'False'} : Bool := FALSE;   // I557.0
      "I557.1" { ExternalVisible := 'False'} : Bool := FALSE;   // I557.1
      "I557.2" { ExternalVisible := 'False'} : Bool := FALSE;   // I557.2
      "I557.3" { ExternalVisible := 'False'} : Bool := FALSE;   // I557.3
      "I557.4" { ExternalVisible := 'False'} : Bool := FALSE;   // I557.4
      "I557.5" { ExternalVisible := 'False'} : Bool := FALSE;   // I557.5
      "I557.6" { ExternalVisible := 'False'} : Bool := FALSE;   // I557.6
      "I557.7" { ExternalVisible := 'False'} : Bool := FALSE;   // I557.7
      "I558.0" { ExternalVisible := 'False'} : Bool := FALSE;   // I558.0
      "I558.1" { ExternalVisible := 'False'} : Bool := FALSE;   // I558.1
      "I558.2" { ExternalVisible := 'False'} : Bool := FALSE;   // I558.2
      "I558.3" { ExternalVisible := 'False'} : Bool := FALSE;   // I558.3
      "I558.4" { ExternalVisible := 'False'} : Bool := FALSE;   // I558.4
      "I558.5" { ExternalVisible := 'False'} : Bool := FALSE;   // I558.5
      "I558.6" { ExternalVisible := 'False'} : Bool := FALSE;   // I558.6
      "I558.7" { ExternalVisible := 'False'} : Bool := FALSE;   // I558.7
      "I559.0" { ExternalVisible := 'False'} : Bool := FALSE;   // I559.0
      "I559.1" { ExternalVisible := 'False'} : Bool := FALSE;   // I559.1
      "I559.2" { ExternalVisible := 'False'} : Bool := FALSE;   // I559.2
      "I559.3" { ExternalVisible := 'False'} : Bool := FALSE;   // I559.3
      "I559.4" { ExternalVisible := 'False'} : Bool := FALSE;   // I559.4
      "I559.5" { ExternalVisible := 'False'} : Bool := FALSE;   // I559.5
      "I559.6" { ExternalVisible := 'False'} : Bool := FALSE;   // I559.6
      "I559.7" { ExternalVisible := 'False'} : Bool := FALSE;   // I559.7
      "I560.0" { ExternalVisible := 'False'} : Bool := FALSE;   // I560.0
      "I560.1" { ExternalVisible := 'False'} : Bool := FALSE;   // I560.1
      "I560.2" { ExternalVisible := 'False'} : Bool := FALSE;   // I560.2
      "I560.3" { ExternalVisible := 'False'} : Bool := FALSE;   // I560.3
      "I560.4" { ExternalVisible := 'False'} : Bool := FALSE;   // I560.4
      "I560.5" { ExternalVisible := 'False'} : Bool := FALSE;   // I560.5
      "I560.6" { ExternalVisible := 'False'} : Bool := FALSE;   // I560.6
      "I560.7" { ExternalVisible := 'False'} : Bool := FALSE;   // I560.7
      "I561.0" { ExternalVisible := 'False'} : Bool := FALSE;   // I561.0
      "I561.1" { ExternalVisible := 'False'} : Bool := FALSE;   // I561.1
      "I561.2" { ExternalVisible := 'False'} : Bool := FALSE;   // I561.2
      "I561.3" { ExternalVisible := 'False'} : Bool := FALSE;   // I561.3
      "I561.4" { ExternalVisible := 'False'} : Bool := FALSE;   // I561.4
      "I561.5" { ExternalVisible := 'False'} : Bool := FALSE;   // I561.5
      "I561.6" { ExternalVisible := 'False'} : Bool := FALSE;   // I561.6
      "I561.7" { ExternalVisible := 'False'} : Bool := FALSE;   // I561.7
      "I562.0" { ExternalVisible := 'False'} : Bool := FALSE;   // I562.0
      "I562.1" { ExternalVisible := 'False'} : Bool := FALSE;   // I562.1
      "I562.2" { ExternalVisible := 'False'} : Bool := FALSE;   // I562.2
      "I562.3" { ExternalVisible := 'False'} : Bool := FALSE;   // I562.3
      "I562.4" { ExternalVisible := 'False'} : Bool := FALSE;   // I562.4
      "I562.5" { ExternalVisible := 'False'} : Bool := FALSE;   // I562.5
      "I562.6" { ExternalVisible := 'False'} : Bool := FALSE;   // I562.6
      "I562.7" { ExternalVisible := 'False'} : Bool := FALSE;   // I562.7
      "I563.0" { ExternalVisible := 'False'} : Bool := FALSE;   // I563.0
      "I563.1" { ExternalVisible := 'False'} : Bool := FALSE;   // I563.1
      "I563.2" { ExternalVisible := 'False'} : Bool := FALSE;   // I563.2
      "I563.3" { ExternalVisible := 'False'} : Bool := FALSE;   // I563.3
      "I563.4" { ExternalVisible := 'False'} : Bool := FALSE;   // I563.4
      "I563.5" { ExternalVisible := 'False'} : Bool := FALSE;   // I563.5
      "I563.6" { ExternalVisible := 'False'} : Bool := FALSE;   // I563.6
      "I563.7" { ExternalVisible := 'False'} : Bool := FALSE;   // I563.7
      "I564.0" { ExternalVisible := 'False'} : Bool := FALSE;   // I564.0
      "I564.1" { ExternalVisible := 'False'} : Bool := FALSE;   // I564.1
      "I564.2" { ExternalVisible := 'False'} : Bool := FALSE;   // I564.2
      "I564.3" { ExternalVisible := 'False'} : Bool := FALSE;   // I564.3
      "I564.4" { ExternalVisible := 'False'} : Bool := FALSE;   // I564.4
      "I564.5" { ExternalVisible := 'False'} : Bool := FALSE;   // I564.5
      "I564.6" { ExternalVisible := 'False'} : Bool := FALSE;   // I564.6
      "I564.7" { ExternalVisible := 'False'} : Bool := FALSE;   // I564.7
      "I565.0" { ExternalVisible := 'False'} : Bool := FALSE;   // I565.0
      "I565.1" { ExternalVisible := 'False'} : Bool := FALSE;   // I565.1
      "I565.2" { ExternalVisible := 'False'} : Bool := FALSE;   // I565.2
      "I565.3" { ExternalVisible := 'False'} : Bool := FALSE;   // I565.3
      "I565.4" { ExternalVisible := 'False'} : Bool := FALSE;   // I565.4
      "I565.5" { ExternalVisible := 'False'} : Bool := FALSE;   // I565.5
      "I565.6" { ExternalVisible := 'False'} : Bool := FALSE;   // I565.6
      "I565.7" { ExternalVisible := 'False'} : Bool := FALSE;   // I565.7
      "I566.0" { ExternalVisible := 'False'} : Bool := FALSE;   // I566.0
      "I566.1" { ExternalVisible := 'False'} : Bool := FALSE;   // I566.1
      "I566.2" { ExternalVisible := 'False'} : Bool := FALSE;   // I566.2
      "I566.3" { ExternalVisible := 'False'} : Bool := FALSE;   // I566.3
      "I566.4" { ExternalVisible := 'False'} : Bool := FALSE;   // I566.4
      "I566.5" { ExternalVisible := 'False'} : Bool := FALSE;   // I566.5
      "I566.6" { ExternalVisible := 'False'} : Bool := FALSE;   // I566.6
      "I566.7" { ExternalVisible := 'False'} : Bool := FALSE;   // I566.7
      "I567.0" { ExternalVisible := 'False'} : Bool := FALSE;   // I567.0
      "I567.1" { ExternalVisible := 'False'} : Bool := FALSE;   // I567.1
      "I567.2" { ExternalVisible := 'False'} : Bool := FALSE;   // I567.2
      "I567.3" { ExternalVisible := 'False'} : Bool := FALSE;   // I567.3
      "I567.4" { ExternalVisible := 'False'} : Bool := FALSE;   // I567.4
      "I567.5" { ExternalVisible := 'False'} : Bool := FALSE;   // I567.5
      "I567.6" { ExternalVisible := 'False'} : Bool := FALSE;   // I567.6
      "I567.7" { ExternalVisible := 'False'} : Bool := FALSE;   // I567.7
      "I568.0" { ExternalVisible := 'False'} : Bool := FALSE;   // I568.0
      "I568.1" { ExternalVisible := 'False'} : Bool := FALSE;   // I568.1
      "I568.2" { ExternalVisible := 'False'} : Bool := FALSE;   // I568.2
      "I568.3" { ExternalVisible := 'False'} : Bool := FALSE;   // I568.3
      "I568.4" { ExternalVisible := 'False'} : Bool := FALSE;   // I568.4
      "I568.5" { ExternalVisible := 'False'} : Bool := FALSE;   // I568.5
      "I568.6" { ExternalVisible := 'False'} : Bool := FALSE;   // I568.6
      "I568.7" { ExternalVisible := 'False'} : Bool := FALSE;   // I568.7
      "I569.0" { ExternalVisible := 'False'} : Bool := FALSE;   // I569.0
      "I569.1" { ExternalVisible := 'False'} : Bool := FALSE;   // I569.1
      "I569.2" { ExternalVisible := 'False'} : Bool := FALSE;   // I569.2
      "I569.3" { ExternalVisible := 'False'} : Bool := FALSE;   // I569.3
      "I569.4" { ExternalVisible := 'False'} : Bool := FALSE;   // I569.4
      "I569.5" { ExternalVisible := 'False'} : Bool := FALSE;   // I569.5
      "I569.6" { ExternalVisible := 'False'} : Bool := FALSE;   // I569.6
      "I569.7" { ExternalVisible := 'False'} : Bool := FALSE;   // I569.7
      "I570.0" { ExternalVisible := 'False'} : Bool := FALSE;   // I570.0
      "I570.1" { ExternalVisible := 'False'} : Bool := FALSE;   // I570.1
      "I570.2" { ExternalVisible := 'False'} : Bool := FALSE;   // I570.2
      "I570.3" { ExternalVisible := 'False'} : Bool := FALSE;   // I570.3
      "I570.4" { ExternalVisible := 'False'} : Bool := FALSE;   // I570.4
      "I570.5" { ExternalVisible := 'False'} : Bool := FALSE;   // I570.5
      "I570.6" { ExternalVisible := 'False'} : Bool := FALSE;   // I570.6
      "I570.7" { ExternalVisible := 'False'} : Bool := FALSE;   // I570.7
      "I571.0" { ExternalVisible := 'False'} : Bool := FALSE;   // I571.0
      "I571.1" { ExternalVisible := 'False'} : Bool := FALSE;   // I571.1
      "I571.2" { ExternalVisible := 'False'} : Bool := FALSE;   // I571.2
      "I571.3" { ExternalVisible := 'False'} : Bool := FALSE;   // I571.3
      "I571.4" { ExternalVisible := 'False'} : Bool := FALSE;   // I571.4
      "I571.5" { ExternalVisible := 'False'} : Bool := FALSE;   // I571.5
      "I571.6" { ExternalVisible := 'False'} : Bool := FALSE;   // I571.6
      "I571.7" { ExternalVisible := 'False'} : Bool := FALSE;   // I571.7
      "I572.0" { ExternalVisible := 'False'} : Bool := FALSE;   // I572.0
      "I572.1" { ExternalVisible := 'False'} : Bool := FALSE;   // I572.1
      "I572.2" { ExternalVisible := 'False'} : Bool := FALSE;   // I572.2
      "I572.3" { ExternalVisible := 'False'} : Bool := FALSE;   // I572.3
      "I572.4" { ExternalVisible := 'False'} : Bool := FALSE;   // I572.4
      "I572.5" { ExternalVisible := 'False'} : Bool := FALSE;   // I572.5
      "I572.6" { ExternalVisible := 'False'} : Bool := FALSE;   // I572.6
      "I572.7" { ExternalVisible := 'False'} : Bool := FALSE;   // I572.7
      "I573.0" { ExternalVisible := 'False'} : Bool := FALSE;   // I573.0
      "I573.1" { ExternalVisible := 'False'} : Bool := FALSE;   // I573.1
      "I573.2" { ExternalVisible := 'False'} : Bool := FALSE;   // I573.2
      "I573.3" { ExternalVisible := 'False'} : Bool := FALSE;   // I573.3
      "I573.4" { ExternalVisible := 'False'} : Bool := FALSE;   // I573.4
      "I573.5" { ExternalVisible := 'False'} : Bool := FALSE;   // I573.5
      "I573.6" { ExternalVisible := 'False'} : Bool := FALSE;   // I573.6
      "I573.7" { ExternalVisible := 'False'} : Bool := FALSE;   // I573.7
      "I574.0" { ExternalVisible := 'False'} : Bool := FALSE;   // I574.0
      "I574.1" { ExternalVisible := 'False'} : Bool := FALSE;   // I574.1
      "I574.2" { ExternalVisible := 'False'} : Bool := FALSE;   // I574.2
      "I574.3" { ExternalVisible := 'False'} : Bool := FALSE;   // I574.3
      "I574.4" { ExternalVisible := 'False'} : Bool := FALSE;   // I574.4
      "I574.5" { ExternalVisible := 'False'} : Bool := FALSE;   // I574.5
      "I574.6" { ExternalVisible := 'False'} : Bool := FALSE;   // I574.6
      "I574.7" { ExternalVisible := 'False'} : Bool := FALSE;   // I574.7
      "I575.0" { ExternalVisible := 'False'} : Bool := FALSE;   // I575.0
      "I575.1" { ExternalVisible := 'False'} : Bool := FALSE;   // I575.1
      "I575.2" { ExternalVisible := 'False'} : Bool := FALSE;   // I575.2
      "I575.3" { ExternalVisible := 'False'} : Bool := FALSE;   // I575.3
      "I575.4" { ExternalVisible := 'False'} : Bool := FALSE;   // I575.4
      "I575.5" { ExternalVisible := 'False'} : Bool := FALSE;   // I575.5
      "I575.6" { ExternalVisible := 'False'} : Bool := FALSE;   // I575.6
      "I575.7" { ExternalVisible := 'False'} : Bool := FALSE;   // I575.7
      "I576.0" { ExternalVisible := 'False'} : Bool := FALSE;   // I576.0
      "I576.1" { ExternalVisible := 'False'} : Bool := FALSE;   // I576.1
      "I576.2" { ExternalVisible := 'False'} : Bool := FALSE;   // I576.2
      "I576.3" { ExternalVisible := 'False'} : Bool := FALSE;   // I576.3
      "I576.4" { ExternalVisible := 'False'} : Bool := FALSE;   // I576.4
      "I576.5" { ExternalVisible := 'False'} : Bool := FALSE;   // I576.5
      "I576.6" { ExternalVisible := 'False'} : Bool := FALSE;   // I576.6
      "I576.7" { ExternalVisible := 'False'} : Bool := FALSE;   // I576.7
      "I577.0" { ExternalVisible := 'False'} : Bool := FALSE;   // I577.0
      "I577.1" { ExternalVisible := 'False'} : Bool := FALSE;   // I577.1
      "I577.2" { ExternalVisible := 'False'} : Bool := FALSE;   // I577.2
      "I577.3" { ExternalVisible := 'False'} : Bool := FALSE;   // I577.3
      "I577.4" { ExternalVisible := 'False'} : Bool := FALSE;   // I577.4
      "I577.5" { ExternalVisible := 'False'} : Bool := FALSE;   // I577.5
      "I577.6" { ExternalVisible := 'False'} : Bool := FALSE;   // I577.6
      "I577.7" { ExternalVisible := 'False'} : Bool := FALSE;   // I577.7
      "I578.0" { ExternalVisible := 'False'} : Bool := FALSE;   // I578.0
      "I578.1" { ExternalVisible := 'False'} : Bool := FALSE;   // I578.1
      "I578.2" { ExternalVisible := 'False'} : Bool := FALSE;   // I578.2
      "I578.3" { ExternalVisible := 'False'} : Bool := FALSE;   // I578.3
      "I578.4" { ExternalVisible := 'False'} : Bool := FALSE;   // I578.4
      "I578.5" { ExternalVisible := 'False'} : Bool := FALSE;   // I578.5
      "I578.6" { ExternalVisible := 'False'} : Bool := FALSE;   // I578.6
      "I578.7" { ExternalVisible := 'False'} : Bool := FALSE;   // I578.7
      "I579.0" { ExternalVisible := 'False'} : Bool := FALSE;   // I579.0
      "I579.1" { ExternalVisible := 'False'} : Bool := FALSE;   // I579.1
      "I579.2" { ExternalVisible := 'False'} : Bool := FALSE;   // I579.2
      "I579.3" { ExternalVisible := 'False'} : Bool := FALSE;   // I579.3
      "I579.4" { ExternalVisible := 'False'} : Bool := FALSE;   // I579.4
      "I579.5" { ExternalVisible := 'False'} : Bool := FALSE;   // I579.5
      "I579.6" { ExternalVisible := 'False'} : Bool := FALSE;   // I579.6
      "I579.7" { ExternalVisible := 'False'} : Bool := FALSE;   // I579.7
      "I580.0" { ExternalVisible := 'False'} : Bool := FALSE;   // I580.0
      "I580.1" { ExternalVisible := 'False'} : Bool := FALSE;   // I580.1
      "I580.2" { ExternalVisible := 'False'} : Bool := FALSE;   // I580.2
      "I580.3" { ExternalVisible := 'False'} : Bool := FALSE;   // I580.3
      "I580.4" { ExternalVisible := 'False'} : Bool := FALSE;   // I580.4
      "I580.5" { ExternalVisible := 'False'} : Bool := FALSE;   // I580.5
      "I580.6" { ExternalVisible := 'False'} : Bool := FALSE;   // I580.6
      "I580.7" { ExternalVisible := 'False'} : Bool := FALSE;   // I580.7
      "I581.0" { ExternalVisible := 'False'} : Bool := FALSE;   // I581.0
      "I581.1" { ExternalVisible := 'False'} : Bool := FALSE;   // I581.1
      "I581.2" { ExternalVisible := 'False'} : Bool := FALSE;   // I581.2
      "I581.3" { ExternalVisible := 'False'} : Bool := FALSE;   // I581.3
      "I581.4" { ExternalVisible := 'False'} : Bool := FALSE;   // I581.4
      "I581.5" { ExternalVisible := 'False'} : Bool := FALSE;   // I581.5
      "I581.6" { ExternalVisible := 'False'} : Bool := FALSE;   // I581.6
      "I581.7" { ExternalVisible := 'False'} : Bool := FALSE;   // I581.7
      "I582.0" { ExternalVisible := 'False'} : Bool := FALSE;   // I582.0
      "I582.1" { ExternalVisible := 'False'} : Bool := FALSE;   // I582.1
      "I582.2" { ExternalVisible := 'False'} : Bool := FALSE;   // I582.2
      "I582.3" { ExternalVisible := 'False'} : Bool := FALSE;   // I582.3
      "I582.4" { ExternalVisible := 'False'} : Bool := FALSE;   // I582.4
      "I582.5" { ExternalVisible := 'False'} : Bool := FALSE;   // I582.5
      "I582.6" { ExternalVisible := 'False'} : Bool := FALSE;   // I582.6
      "I582.7" { ExternalVisible := 'False'} : Bool := FALSE;   // I582.7
      "I583.0" { ExternalVisible := 'False'} : Bool := FALSE;   // I583.0
      "I583.1" { ExternalVisible := 'False'} : Bool := FALSE;   // I583.1
      "I583.2" { ExternalVisible := 'False'} : Bool := FALSE;   // I583.2
      "I583.3" { ExternalVisible := 'False'} : Bool := FALSE;   // I583.3
      "I583.4" { ExternalVisible := 'False'} : Bool := FALSE;   // I583.4
      "I583.5" { ExternalVisible := 'False'} : Bool := FALSE;   // I583.5
      "I583.6" { ExternalVisible := 'False'} : Bool := FALSE;   // I583.6
      "I583.7" { ExternalVisible := 'False'} : Bool := FALSE;   // I583.7
      "I584.0" { ExternalVisible := 'False'} : Bool := FALSE;   // I584.0
      "I584.1" { ExternalVisible := 'False'} : Bool := FALSE;   // I584.1
      "I584.2" { ExternalVisible := 'False'} : Bool := FALSE;   // I584.2
      "I584.3" { ExternalVisible := 'False'} : Bool := FALSE;   // I584.3
      "I584.4" { ExternalVisible := 'False'} : Bool := FALSE;   // I584.4
      "I584.5" { ExternalVisible := 'False'} : Bool := FALSE;   // I584.5
      "I584.6" { ExternalVisible := 'False'} : Bool := FALSE;   // I584.6
      "I584.7" { ExternalVisible := 'False'} : Bool := FALSE;   // I584.7
      "I585.0" { ExternalVisible := 'False'} : Bool := FALSE;   // I585.0
      "I585.1" { ExternalVisible := 'False'} : Bool := FALSE;   // I585.1
      "I585.2" { ExternalVisible := 'False'} : Bool := FALSE;   // I585.2
      "I585.3" { ExternalVisible := 'False'} : Bool := FALSE;   // I585.3
      "I585.4" { ExternalVisible := 'False'} : Bool := FALSE;   // I585.4
      "I585.5" { ExternalVisible := 'False'} : Bool := FALSE;   // I585.5
      "I585.6" { ExternalVisible := 'False'} : Bool := FALSE;   // I585.6
      "I585.7" { ExternalVisible := 'False'} : Bool := FALSE;   // I585.7
      "I586.0" { ExternalVisible := 'False'} : Bool := FALSE;   // I586.0
      "I586.1" { ExternalVisible := 'False'} : Bool := FALSE;   // I586.1
      "I586.2" { ExternalVisible := 'False'} : Bool := FALSE;   // I586.2
      "I586.3" { ExternalVisible := 'False'} : Bool := FALSE;   // I586.3
      "I586.4" { ExternalVisible := 'False'} : Bool := FALSE;   // I586.4
      "I586.5" { ExternalVisible := 'False'} : Bool := FALSE;   // I586.5
      "I586.6" { ExternalVisible := 'False'} : Bool := FALSE;   // I586.6
      "I586.7" { ExternalVisible := 'False'} : Bool := FALSE;   // I586.7
      "I587.0" { ExternalVisible := 'False'} : Bool := FALSE;   // I587.0
      "I587.1" { ExternalVisible := 'False'} : Bool := FALSE;   // I587.1
      "I587.2" { ExternalVisible := 'False'} : Bool := FALSE;   // I587.2
      "I587.3" { ExternalVisible := 'False'} : Bool := FALSE;   // I587.3
      "I587.4" { ExternalVisible := 'False'} : Bool := FALSE;   // I587.4
      "I587.5" { ExternalVisible := 'False'} : Bool := FALSE;   // I587.5
      "I587.6" { ExternalVisible := 'False'} : Bool := FALSE;   // I587.6
      "I587.7" { ExternalVisible := 'False'} : Bool := FALSE;   // I587.7
      "I588.0" { ExternalVisible := 'False'} : Bool := FALSE;   // I588.0
      "I588.1" { ExternalVisible := 'False'} : Bool := FALSE;   // I588.1
      "I588.2" { ExternalVisible := 'False'} : Bool := FALSE;   // I588.2
      "I588.3" { ExternalVisible := 'False'} : Bool := FALSE;   // I588.3
      "I588.4" { ExternalVisible := 'False'} : Bool := FALSE;   // I588.4
      "I588.5" { ExternalVisible := 'False'} : Bool := FALSE;   // I588.5
      "I588.6" { ExternalVisible := 'False'} : Bool := FALSE;   // I588.6
      "I588.7" { ExternalVisible := 'False'} : Bool := FALSE;   // I588.7
      "I589.0" { ExternalVisible := 'False'} : Bool := FALSE;   // I589.0
      "I589.1" { ExternalVisible := 'False'} : Bool := FALSE;   // I589.1
      "I589.2" { ExternalVisible := 'False'} : Bool := FALSE;   // I589.2
      "I589.3" { ExternalVisible := 'False'} : Bool := FALSE;   // I589.3
      "I589.4" { ExternalVisible := 'False'} : Bool := FALSE;   // I589.4
      "I589.5" { ExternalVisible := 'False'} : Bool := FALSE;   // I589.5
      "I589.6" { ExternalVisible := 'False'} : Bool := FALSE;   // I589.6
      "I589.7" { ExternalVisible := 'False'} : Bool := FALSE;   // I589.7
      "I590.0" { ExternalVisible := 'False'} : Bool := FALSE;   // I590.0
      "I590.1" { ExternalVisible := 'False'} : Bool := FALSE;   // I590.1
      "I590.2" { ExternalVisible := 'False'} : Bool := FALSE;   // I590.2
      "I590.3" { ExternalVisible := 'False'} : Bool := FALSE;   // I590.3
      "I590.4" { ExternalVisible := 'False'} : Bool := FALSE;   // I590.4
      "I590.5" { ExternalVisible := 'False'} : Bool := FALSE;   // I590.5
      "I590.6" { ExternalVisible := 'False'} : Bool := FALSE;   // I590.6
      "I590.7" { ExternalVisible := 'False'} : Bool := FALSE;   // I590.7
      "I591.0" { ExternalVisible := 'False'} : Bool := FALSE;   // I591.0
      "I591.1" { ExternalVisible := 'False'} : Bool := FALSE;   // I591.1
      "I591.2" { ExternalVisible := 'False'} : Bool := FALSE;   // I591.2
      "I591.3" { ExternalVisible := 'False'} : Bool := FALSE;   // I591.3
      "I591.4" { ExternalVisible := 'False'} : Bool := FALSE;   // I591.4
      "I591.5" { ExternalVisible := 'False'} : Bool := FALSE;   // I591.5
      "I591.6" { ExternalVisible := 'False'} : Bool := FALSE;   // I591.6
      "I591.7" { ExternalVisible := 'False'} : Bool := FALSE;   // I591.7
      "I592.0" { ExternalVisible := 'False'} : Bool := FALSE;   // I592.0
      "I592.1" { ExternalVisible := 'False'} : Bool := FALSE;   // I592.1
      "I592.2" { ExternalVisible := 'False'} : Bool := FALSE;   // I592.2
      "I592.3" { ExternalVisible := 'False'} : Bool := FALSE;   // I592.3
      "I592.4" { ExternalVisible := 'False'} : Bool := FALSE;   // I592.4
      "I592.5" { ExternalVisible := 'False'} : Bool := FALSE;   // I592.5
      "I592.6" { ExternalVisible := 'False'} : Bool := FALSE;   // I592.6
      "I592.7" { ExternalVisible := 'False'} : Bool := FALSE;   // I592.7
      "I593.0" { ExternalVisible := 'False'} : Bool := FALSE;   // I593.0
      "I593.1" { ExternalVisible := 'False'} : Bool := FALSE;   // I593.1
      "I593.2" { ExternalVisible := 'False'} : Bool := FALSE;   // I593.2
      "I593.3" { ExternalVisible := 'False'} : Bool := FALSE;   // I593.3
      "I593.4" { ExternalVisible := 'False'} : Bool := FALSE;   // I593.4
      "I593.5" { ExternalVisible := 'False'} : Bool := FALSE;   // I593.5
      "I593.6" { ExternalVisible := 'False'} : Bool := FALSE;   // I593.6
      "I593.7" { ExternalVisible := 'False'} : Bool := FALSE;   // I593.7
      "I594.0" { ExternalVisible := 'False'} : Bool := FALSE;   // I594.0
      "I594.1" { ExternalVisible := 'False'} : Bool := FALSE;   // I594.1
      "I594.2" { ExternalVisible := 'False'} : Bool := FALSE;   // I594.2
      "I594.3" { ExternalVisible := 'False'} : Bool := FALSE;   // I594.3
      "I594.4" { ExternalVisible := 'False'} : Bool := FALSE;   // I594.4
      "I594.5" { ExternalVisible := 'False'} : Bool := FALSE;   // I594.5
      "I594.6" { ExternalVisible := 'False'} : Bool := FALSE;   // I594.6
      "I594.7" { ExternalVisible := 'False'} : Bool := FALSE;   // I594.7
      "I595.0" { ExternalVisible := 'False'} : Bool := FALSE;   // I595.0
      "I595.1" { ExternalVisible := 'False'} : Bool := FALSE;   // I595.1
      "I595.2" { ExternalVisible := 'False'} : Bool := FALSE;   // I595.2
      "I595.3" { ExternalVisible := 'False'} : Bool := FALSE;   // I595.3
      "I595.4" { ExternalVisible := 'False'} : Bool := FALSE;   // I595.4
      "I595.5" { ExternalVisible := 'False'} : Bool := FALSE;   // I595.5
      "I595.6" { ExternalVisible := 'False'} : Bool := FALSE;   // I595.6
      "I595.7" { ExternalVisible := 'False'} : Bool := FALSE;   // I595.7
      "I596.0" { ExternalVisible := 'False'} : Bool := FALSE;   // I596.0
      "I596.1" { ExternalVisible := 'False'} : Bool := FALSE;   // I596.1
      "I596.2" { ExternalVisible := 'False'} : Bool := FALSE;   // I596.2
      "I596.3" { ExternalVisible := 'False'} : Bool := FALSE;   // I596.3
      "I596.4" { ExternalVisible := 'False'} : Bool := FALSE;   // I596.4
      "I596.5" { ExternalVisible := 'False'} : Bool := FALSE;   // I596.5
      "I596.6" { ExternalVisible := 'False'} : Bool := FALSE;   // I596.6
      "I596.7" { ExternalVisible := 'False'} : Bool := FALSE;   // I596.7
      "I597.0" { ExternalVisible := 'False'} : Bool := FALSE;   // I597.0
      "I597.1" { ExternalVisible := 'False'} : Bool := FALSE;   // I597.1
      "I597.2" { ExternalVisible := 'False'} : Bool := FALSE;   // I597.2
      "I597.3" { ExternalVisible := 'False'} : Bool := FALSE;   // I597.3
      "I597.4" { ExternalVisible := 'False'} : Bool := FALSE;   // I597.4
      "I597.5" { ExternalVisible := 'False'} : Bool := FALSE;   // I597.5
      "I597.6" { ExternalVisible := 'False'} : Bool := FALSE;   // I597.6
      "I597.7" { ExternalVisible := 'False'} : Bool := FALSE;   // I597.7
      "I598.0" { ExternalVisible := 'False'} : Bool := FALSE;   // I598.0
      "I598.1" { ExternalVisible := 'False'} : Bool := FALSE;   // I598.1
      "I598.2" { ExternalVisible := 'False'} : Bool := FALSE;   // I598.2
      "I598.3" { ExternalVisible := 'False'} : Bool := FALSE;   // I598.3
      "I598.4" { ExternalVisible := 'False'} : Bool := FALSE;   // I598.4
      "I598.5" { ExternalVisible := 'False'} : Bool := FALSE;   // I598.5
      "I598.6" { ExternalVisible := 'False'} : Bool := FALSE;   // I598.6
      "I598.7" { ExternalVisible := 'False'} : Bool := FALSE;   // I598.7
      "I599.0" { ExternalVisible := 'False'} : Bool := FALSE;   // I599.0
      "I599.1" { ExternalVisible := 'False'} : Bool := FALSE;   // I599.1
      "I599.2" { ExternalVisible := 'False'} : Bool := FALSE;   // I599.2
      "I599.3" { ExternalVisible := 'False'} : Bool := FALSE;   // I599.3
      "I599.4" { ExternalVisible := 'False'} : Bool := FALSE;   // I599.4
      "I599.5" { ExternalVisible := 'False'} : Bool := FALSE;   // I599.5
      "I599.6" { ExternalVisible := 'False'} : Bool := FALSE;   // I599.6
      "I599.7" { ExternalVisible := 'False'} : Bool := FALSE;   // I599.7
      "I600.0" { ExternalVisible := 'False'} : Bool := FALSE;   // I600.0
      "I600.1" { ExternalVisible := 'False'} : Bool := FALSE;   // I600.1
      "I600.2" { ExternalVisible := 'False'} : Bool := FALSE;   // I600.2
      "I600.3" { ExternalVisible := 'False'} : Bool := FALSE;   // I600.3
      "I600.4" { ExternalVisible := 'False'} : Bool := FALSE;   // I600.4
      "I600.5" { ExternalVisible := 'False'} : Bool := FALSE;   // I600.5
      "I600.6" { ExternalVisible := 'False'} : Bool := FALSE;   // I600.6
      "I600.7" { ExternalVisible := 'False'} : Bool := FALSE;   // I600.7
      "I601.0" { ExternalVisible := 'False'} : Bool := FALSE;   // I601.0
      "I601.1" { ExternalVisible := 'False'} : Bool := FALSE;   // I601.1
      "I601.2" { ExternalVisible := 'False'} : Bool := FALSE;   // I601.2
      "I601.3" { ExternalVisible := 'False'} : Bool := FALSE;   // I601.3
      "I601.4" { ExternalVisible := 'False'} : Bool := FALSE;   // I601.4
      "I601.5" { ExternalVisible := 'False'} : Bool := FALSE;   // I601.5
      "I601.6" { ExternalVisible := 'False'} : Bool := FALSE;   // I601.6
      "I601.7" { ExternalVisible := 'False'} : Bool := FALSE;   // I601.7
      "I602.0" { ExternalVisible := 'False'} : Bool := FALSE;   // I602.0
      "I602.1" { ExternalVisible := 'False'} : Bool := FALSE;   // I602.1
      "I602.2" { ExternalVisible := 'False'} : Bool := FALSE;   // I602.2
      "I602.3" { ExternalVisible := 'False'} : Bool := FALSE;   // I602.3
      "I602.4" { ExternalVisible := 'False'} : Bool := FALSE;   // I602.4
      "I602.5" { ExternalVisible := 'False'} : Bool := FALSE;   // I602.5
      "I602.6" { ExternalVisible := 'False'} : Bool := FALSE;   // I602.6
      "I602.7" { ExternalVisible := 'False'} : Bool := FALSE;   // I602.7
      "I603.0" { ExternalVisible := 'False'} : Bool := FALSE;   // I603.0
      "I603.1" { ExternalVisible := 'False'} : Bool := FALSE;   // I603.1
      "I603.2" { ExternalVisible := 'False'} : Bool := FALSE;   // I603.2
      "I603.3" { ExternalVisible := 'False'} : Bool := FALSE;   // I603.3
      "I603.4" { ExternalVisible := 'False'} : Bool := FALSE;   // I603.4
      "I603.5" { ExternalVisible := 'False'} : Bool := FALSE;   // I603.5
      "I603.6" { ExternalVisible := 'False'} : Bool := FALSE;   // I603.6
      "I603.7" { ExternalVisible := 'False'} : Bool := FALSE;   // I603.7
      "I604.0" { ExternalVisible := 'False'} : Bool := FALSE;   // I604.0
      "I604.1" { ExternalVisible := 'False'} : Bool := FALSE;   // I604.1
      "I604.2" { ExternalVisible := 'False'} : Bool := FALSE;   // I604.2
      "I604.3" { ExternalVisible := 'False'} : Bool := FALSE;   // I604.3
      "I604.4" { ExternalVisible := 'False'} : Bool := FALSE;   // I604.4
      "I604.5" { ExternalVisible := 'False'} : Bool := FALSE;   // I604.5
      "I604.6" { ExternalVisible := 'False'} : Bool := FALSE;   // I604.6
      "I604.7" { ExternalVisible := 'False'} : Bool := FALSE;   // I604.7
      "I605.0" { ExternalVisible := 'False'} : Bool := FALSE;   // I605.0
      "I605.1" { ExternalVisible := 'False'} : Bool := FALSE;   // I605.1
      "I605.2" { ExternalVisible := 'False'} : Bool := FALSE;   // I605.2
      "I605.3" { ExternalVisible := 'False'} : Bool := FALSE;   // I605.3
      "I605.4" { ExternalVisible := 'False'} : Bool := FALSE;   // I605.4
      "I605.5" { ExternalVisible := 'False'} : Bool := FALSE;   // I605.5
      "I605.6" { ExternalVisible := 'False'} : Bool := FALSE;   // I605.6
      "I605.7" { ExternalVisible := 'False'} : Bool := FALSE;   // I605.7
      "I606.0" { ExternalVisible := 'False'} : Bool := FALSE;   // I606.0
      "I606.1" { ExternalVisible := 'False'} : Bool := FALSE;   // I606.1
      "I606.2" { ExternalVisible := 'False'} : Bool := FALSE;   // I606.2
      "I606.3" { ExternalVisible := 'False'} : Bool := FALSE;   // I606.3
      "I606.4" { ExternalVisible := 'False'} : Bool := FALSE;   // I606.4
      "I606.5" { ExternalVisible := 'False'} : Bool := FALSE;   // I606.5
      "I606.6" { ExternalVisible := 'False'} : Bool := FALSE;   // I606.6
      "I606.7" { ExternalVisible := 'False'} : Bool := FALSE;   // I606.7
      "I607.0" { ExternalVisible := 'False'} : Bool := FALSE;   // I607.0
      "I607.1" { ExternalVisible := 'False'} : Bool := FALSE;   // I607.1
      "I607.2" { ExternalVisible := 'False'} : Bool := FALSE;   // I607.2
      "I607.3" { ExternalVisible := 'False'} : Bool := FALSE;   // I607.3
      "I607.4" { ExternalVisible := 'False'} : Bool := FALSE;   // I607.4
      "I607.5" { ExternalVisible := 'False'} : Bool := FALSE;   // I607.5
      "I607.6" { ExternalVisible := 'False'} : Bool := FALSE;   // I607.6
      "I607.7" { ExternalVisible := 'False'} : Bool := FALSE;   // I607.7
      "I608.0" { ExternalVisible := 'False'} : Bool := FALSE;   // I608.0
      "I608.1" { ExternalVisible := 'False'} : Bool := FALSE;   // I608.1
      "I608.2" { ExternalVisible := 'False'} : Bool := FALSE;   // I608.2
      "I608.3" { ExternalVisible := 'False'} : Bool := FALSE;   // I608.3
      "I608.4" { ExternalVisible := 'False'} : Bool := FALSE;   // I608.4
      "I608.5" { ExternalVisible := 'False'} : Bool := FALSE;   // I608.5
      "I608.6" { ExternalVisible := 'False'} : Bool := FALSE;   // I608.6
      "I608.7" { ExternalVisible := 'False'} : Bool := FALSE;   // I608.7
      "I609.0" { ExternalVisible := 'False'} : Bool := FALSE;   // I609.0
      "I609.1" { ExternalVisible := 'False'} : Bool := FALSE;   // I609.1
      "I609.2" { ExternalVisible := 'False'} : Bool := FALSE;   // I609.2
      "I609.3" { ExternalVisible := 'False'} : Bool := FALSE;   // I609.3
      "I609.4" { ExternalVisible := 'False'} : Bool := FALSE;   // I609.4
      "I609.5" { ExternalVisible := 'False'} : Bool := FALSE;   // I609.5
      "I609.6" { ExternalVisible := 'False'} : Bool := FALSE;   // I609.6
      "I609.7" { ExternalVisible := 'False'} : Bool := FALSE;   // I609.7
      "I610.0" { ExternalVisible := 'False'} : Bool := FALSE;   // I610.0
      "I610.1" { ExternalVisible := 'False'} : Bool := FALSE;   // I610.1
      "I610.2" { ExternalVisible := 'False'} : Bool := FALSE;   // I610.2
      "I610.3" { ExternalVisible := 'False'} : Bool := FALSE;   // I610.3
      "I610.4" { ExternalVisible := 'False'} : Bool := FALSE;   // I610.4
      "I610.5" { ExternalVisible := 'False'} : Bool := FALSE;   // I610.5
      "I610.6" { ExternalVisible := 'False'} : Bool := FALSE;   // I610.6
      "I610.7" { ExternalVisible := 'False'} : Bool := FALSE;   // I610.7
      "I611.0" { ExternalVisible := 'False'} : Bool := FALSE;   // I611.0
      "I611.1" { ExternalVisible := 'False'} : Bool := FALSE;   // I611.1
      "I611.2" { ExternalVisible := 'False'} : Bool := FALSE;   // I611.2
      "I611.3" { ExternalVisible := 'False'} : Bool := FALSE;   // I611.3
      "I611.4" { ExternalVisible := 'False'} : Bool := FALSE;   // I611.4
      "I611.5" { ExternalVisible := 'False'} : Bool := FALSE;   // I611.5
      "I611.6" { ExternalVisible := 'False'} : Bool := FALSE;   // I611.6
      "I611.7" { ExternalVisible := 'False'} : Bool := FALSE;   // I611.7
      "I612.0" { ExternalVisible := 'False'} : Bool := FALSE;   // I612.0
      "I612.1" { ExternalVisible := 'False'} : Bool := FALSE;   // I612.1
      "I612.2" { ExternalVisible := 'False'} : Bool := FALSE;   // I612.2
      "I612.3" { ExternalVisible := 'False'} : Bool := FALSE;   // I612.3
      "I612.4" { ExternalVisible := 'False'} : Bool := FALSE;   // I612.4
      "I612.5" { ExternalVisible := 'False'} : Bool := FALSE;   // I612.5
      "I612.6" { ExternalVisible := 'False'} : Bool := FALSE;   // I612.6
      "I612.7" { ExternalVisible := 'False'} : Bool := FALSE;   // I612.7
      "I613.0" { ExternalVisible := 'False'} : Bool := FALSE;   // I613.0
      "I613.1" { ExternalVisible := 'False'} : Bool := FALSE;   // I613.1
      "I613.2" { ExternalVisible := 'False'} : Bool := FALSE;   // I613.2
      "I613.3" { ExternalVisible := 'False'} : Bool := FALSE;   // I613.3
      "I613.4" { ExternalVisible := 'False'} : Bool := FALSE;   // I613.4
      "I613.5" { ExternalVisible := 'False'} : Bool := FALSE;   // I613.5
      "I613.6" { ExternalVisible := 'False'} : Bool := FALSE;   // I613.6
      "I613.7" { ExternalVisible := 'False'} : Bool := FALSE;   // I613.7
      "I614.0" { ExternalVisible := 'False'} : Bool := FALSE;   // I614.0
      "I614.1" { ExternalVisible := 'False'} : Bool := FALSE;   // I614.1
      "I614.2" { ExternalVisible := 'False'} : Bool := FALSE;   // I614.2
      "I614.3" { ExternalVisible := 'False'} : Bool := FALSE;   // I614.3
      "I614.4" { ExternalVisible := 'False'} : Bool := FALSE;   // I614.4
      "I614.5" { ExternalVisible := 'False'} : Bool := FALSE;   // I614.5
      "I614.6" { ExternalVisible := 'False'} : Bool := FALSE;   // I614.6
      "I614.7" { ExternalVisible := 'False'} : Bool := FALSE;   // I614.7
      "I615.0" { ExternalVisible := 'False'} : Bool := FALSE;   // I615.0
      "I615.1" { ExternalVisible := 'False'} : Bool := FALSE;   // I615.1
      "I615.2" { ExternalVisible := 'False'} : Bool := FALSE;   // I615.2
      "I615.3" { ExternalVisible := 'False'} : Bool := FALSE;   // I615.3
      "I615.4" { ExternalVisible := 'False'} : Bool := FALSE;   // I615.4
      "I615.5" { ExternalVisible := 'False'} : Bool := FALSE;   // I615.5
      "I615.6" { ExternalVisible := 'False'} : Bool := FALSE;   // I615.6
      "I615.7" { ExternalVisible := 'False'} : Bool := FALSE;   // I615.7
      "I616.0" { ExternalVisible := 'False'} : Bool := FALSE;   // I616.0
      "I616.1" { ExternalVisible := 'False'} : Bool := FALSE;   // I616.1
      "I616.2" { ExternalVisible := 'False'} : Bool := FALSE;   // I616.2
      "I616.3" { ExternalVisible := 'False'} : Bool := FALSE;   // I616.3
      "I616.4" { ExternalVisible := 'False'} : Bool := FALSE;   // I616.4
      "I616.5" { ExternalVisible := 'False'} : Bool := FALSE;   // I616.5
      "I616.6" { ExternalVisible := 'False'} : Bool := FALSE;   // I616.6
      "I616.7" { ExternalVisible := 'False'} : Bool := FALSE;   // I616.7
      "I617.0" { ExternalVisible := 'False'} : Bool := FALSE;   // I617.0
      "I617.1" { ExternalVisible := 'False'} : Bool := FALSE;   // I617.1
      "I617.2" { ExternalVisible := 'False'} : Bool := FALSE;   // I617.2
      "I617.3" { ExternalVisible := 'False'} : Bool := FALSE;   // I617.3
      "I617.4" { ExternalVisible := 'False'} : Bool := FALSE;   // I617.4
      "I617.5" { ExternalVisible := 'False'} : Bool := FALSE;   // I617.5
      "I617.6" { ExternalVisible := 'False'} : Bool := FALSE;   // I617.6
      "I617.7" { ExternalVisible := 'False'} : Bool := FALSE;   // I617.7
      "I618.0" { ExternalVisible := 'False'} : Bool := FALSE;   // I618.0
      "I618.1" { ExternalVisible := 'False'} : Bool := FALSE;   // I618.1
      "I618.2" { ExternalVisible := 'False'} : Bool := FALSE;   // I618.2
      "I618.3" { ExternalVisible := 'False'} : Bool := FALSE;   // I618.3
      "I618.4" { ExternalVisible := 'False'} : Bool := FALSE;   // I618.4
      "I618.5" { ExternalVisible := 'False'} : Bool := FALSE;   // I618.5
      "I618.6" { ExternalVisible := 'False'} : Bool := FALSE;   // I618.6
      "I618.7" { ExternalVisible := 'False'} : Bool := FALSE;   // I618.7
      "I619.0" { ExternalVisible := 'False'} : Bool := FALSE;   // I619.0
      "I619.1" { ExternalVisible := 'False'} : Bool := FALSE;   // I619.1
      "I619.2" { ExternalVisible := 'False'} : Bool := FALSE;   // I619.2
      "I619.3" { ExternalVisible := 'False'} : Bool := FALSE;   // I619.3
      "I619.4" { ExternalVisible := 'False'} : Bool := FALSE;   // I619.4
      "I619.5" { ExternalVisible := 'False'} : Bool := FALSE;   // I619.5
      "I619.6" { ExternalVisible := 'False'} : Bool := FALSE;   // I619.6
      "I619.7" { ExternalVisible := 'False'} : Bool := FALSE;   // I619.7
      "I620.0" { ExternalVisible := 'False'} : Bool := FALSE;   // I620.0
      "I620.1" { ExternalVisible := 'False'} : Bool := FALSE;   // I620.1
      "I620.2" { ExternalVisible := 'False'} : Bool := FALSE;   // I620.2
      "I620.3" { ExternalVisible := 'False'} : Bool := FALSE;   // I620.3
      "I620.4" { ExternalVisible := 'False'} : Bool := FALSE;   // I620.4
      "I620.5" { ExternalVisible := 'False'} : Bool := FALSE;   // I620.5
      "I620.6" { ExternalVisible := 'False'} : Bool := FALSE;   // I620.6
      "I620.7" { ExternalVisible := 'False'} : Bool := FALSE;   // I620.7
      "I621.0" { ExternalVisible := 'False'} : Bool := FALSE;   // I621.0
      "I621.1" { ExternalVisible := 'False'} : Bool := FALSE;   // I621.1
      "I621.2" { ExternalVisible := 'False'} : Bool := FALSE;   // I621.2
      "I621.3" { ExternalVisible := 'False'} : Bool := FALSE;   // I621.3
      "I621.4" { ExternalVisible := 'False'} : Bool := FALSE;   // I621.4
      "I621.5" { ExternalVisible := 'False'} : Bool := FALSE;   // I621.5
      "I621.6" { ExternalVisible := 'False'} : Bool := FALSE;   // I621.6
      "I621.7" { ExternalVisible := 'False'} : Bool := FALSE;   // I621.7
      "I622.0" { ExternalVisible := 'False'} : Bool := FALSE;   // I622.0
      "I622.1" { ExternalVisible := 'False'} : Bool := FALSE;   // I622.1
      "I622.2" { ExternalVisible := 'False'} : Bool := FALSE;   // I622.2
      "I622.3" { ExternalVisible := 'False'} : Bool := FALSE;   // I622.3
      "I622.4" { ExternalVisible := 'False'} : Bool := FALSE;   // I622.4
      "I622.5" { ExternalVisible := 'False'} : Bool := FALSE;   // I622.5
      "I622.6" { ExternalVisible := 'False'} : Bool := FALSE;   // I622.6
      "I622.7" { ExternalVisible := 'False'} : Bool := FALSE;   // I622.7
      "I623.0" { ExternalVisible := 'False'} : Bool := FALSE;   // I623.0
      "I623.1" { ExternalVisible := 'False'} : Bool := FALSE;   // I623.1
      "I623.2" { ExternalVisible := 'False'} : Bool := FALSE;   // I623.2
      "I623.3" { ExternalVisible := 'False'} : Bool := FALSE;   // I623.3
      "I623.4" { ExternalVisible := 'False'} : Bool := FALSE;   // I623.4
      "I623.5" { ExternalVisible := 'False'} : Bool := FALSE;   // I623.5
      "I623.6" { ExternalVisible := 'False'} : Bool := FALSE;   // I623.6
      "I623.7" { ExternalVisible := 'False'} : Bool := FALSE;   // I623.7
      "I624.0" { ExternalVisible := 'False'} : Bool := FALSE;   // I624.0
      "I624.1" { ExternalVisible := 'False'} : Bool := FALSE;   // I624.1
      "I624.2" { ExternalVisible := 'False'} : Bool := FALSE;   // I624.2
      "I624.3" { ExternalVisible := 'False'} : Bool := FALSE;   // I624.3
      "I624.4" { ExternalVisible := 'False'} : Bool := FALSE;   // I624.4
      "I624.5" { ExternalVisible := 'False'} : Bool := FALSE;   // I624.5
      "I624.6" { ExternalVisible := 'False'} : Bool := FALSE;   // I624.6
      "I624.7" { ExternalVisible := 'False'} : Bool := FALSE;   // I624.7
      "I625.0" { ExternalVisible := 'False'} : Bool := FALSE;   // I625.0
      "I625.1" { ExternalVisible := 'False'} : Bool := FALSE;   // I625.1
      "I625.2" { ExternalVisible := 'False'} : Bool := FALSE;   // I625.2
      "I625.3" { ExternalVisible := 'False'} : Bool := FALSE;   // I625.3
      "I625.4" { ExternalVisible := 'False'} : Bool := FALSE;   // I625.4
      "I625.5" { ExternalVisible := 'False'} : Bool := FALSE;   // I625.5
      "I625.6" { ExternalVisible := 'False'} : Bool := FALSE;   // I625.6
      "I625.7" { ExternalVisible := 'False'} : Bool := FALSE;   // I625.7
      "I626.0" { ExternalVisible := 'False'} : Bool := FALSE;   // I626.0
      "I626.1" { ExternalVisible := 'False'} : Bool := FALSE;   // I626.1
      "I626.2" { ExternalVisible := 'False'} : Bool := FALSE;   // I626.2
      "I626.3" { ExternalVisible := 'False'} : Bool := FALSE;   // I626.3
      "I626.4" { ExternalVisible := 'False'} : Bool := FALSE;   // I626.4
      "I626.5" { ExternalVisible := 'False'} : Bool := FALSE;   // I626.5
      "I626.6" { ExternalVisible := 'False'} : Bool := FALSE;   // I626.6
      "I626.7" { ExternalVisible := 'False'} : Bool := FALSE;   // I626.7
      "I627.0" { ExternalVisible := 'False'} : Bool := FALSE;   // I627.0
      "I627.1" { ExternalVisible := 'False'} : Bool := FALSE;   // I627.1
      "I627.2" { ExternalVisible := 'False'} : Bool := FALSE;   // I627.2
      "I627.3" { ExternalVisible := 'False'} : Bool := FALSE;   // I627.3
      "I627.4" { ExternalVisible := 'False'} : Bool := FALSE;   // I627.4
      "I627.5" { ExternalVisible := 'False'} : Bool := FALSE;   // I627.5
      "I627.6" { ExternalVisible := 'False'} : Bool := FALSE;   // I627.6
      "I627.7" { ExternalVisible := 'False'} : Bool := FALSE;   // I627.7
      "I628.0" { ExternalVisible := 'False'} : Bool := FALSE;   // I628.0
      "I628.1" { ExternalVisible := 'False'} : Bool := FALSE;   // I628.1
      "I628.2" { ExternalVisible := 'False'} : Bool := FALSE;   // I628.2
      "I628.3" { ExternalVisible := 'False'} : Bool := FALSE;   // I628.3
      "I628.4" { ExternalVisible := 'False'} : Bool := FALSE;   // I628.4
      "I628.5" { ExternalVisible := 'False'} : Bool := FALSE;   // I628.5
      "I628.6" { ExternalVisible := 'False'} : Bool := FALSE;   // I628.6
      "I628.7" { ExternalVisible := 'False'} : Bool := FALSE;   // I628.7
      "I629.0" { ExternalVisible := 'False'} : Bool := FALSE;   // I629.0
      "I629.1" { ExternalVisible := 'False'} : Bool := FALSE;   // I629.1
      "I629.2" { ExternalVisible := 'False'} : Bool := FALSE;   // I629.2
      "I629.3" { ExternalVisible := 'False'} : Bool := FALSE;   // I629.3
      "I629.4" { ExternalVisible := 'False'} : Bool := FALSE;   // I629.4
      "I629.5" { ExternalVisible := 'False'} : Bool := FALSE;   // I629.5
      "I629.6" { ExternalVisible := 'False'} : Bool := FALSE;   // I629.6
      "I629.7" { ExternalVisible := 'False'} : Bool := FALSE;   // I629.7
      "I630.0" { ExternalVisible := 'False'} : Bool := FALSE;   // I630.0
      "I630.1" { ExternalVisible := 'False'} : Bool := FALSE;   // I630.1
      "I630.2" { ExternalVisible := 'False'} : Bool := FALSE;   // I630.2
      "I630.3" { ExternalVisible := 'False'} : Bool := FALSE;   // I630.3
      "I630.4" { ExternalVisible := 'False'} : Bool := FALSE;   // I630.4
      "I630.5" { ExternalVisible := 'False'} : Bool := FALSE;   // I630.5
      "I630.6" { ExternalVisible := 'False'} : Bool := FALSE;   // I630.6
      "I630.7" { ExternalVisible := 'False'} : Bool := FALSE;   // I630.7
      "I631.0" { ExternalVisible := 'False'} : Bool := FALSE;   // I631.0
      "I631.1" { ExternalVisible := 'False'} : Bool := FALSE;   // I631.1
      "I631.2" { ExternalVisible := 'False'} : Bool := FALSE;   // I631.2
      "I631.3" { ExternalVisible := 'False'} : Bool := FALSE;   // I631.3
      "I631.4" { ExternalVisible := 'False'} : Bool := FALSE;   // I631.4
      "I631.5" { ExternalVisible := 'False'} : Bool := FALSE;   // I631.5
      "I631.6" { ExternalVisible := 'False'} : Bool := FALSE;   // I631.6
      "I631.7" { ExternalVisible := 'False'} : Bool := FALSE;   // I631.7
      "I632.0" { ExternalVisible := 'False'} : Bool := FALSE;   // I632.0
      "I632.1" { ExternalVisible := 'False'} : Bool := FALSE;   // I632.1
      "I632.2" { ExternalVisible := 'False'} : Bool := FALSE;   // I632.2
      "I632.3" { ExternalVisible := 'False'} : Bool := FALSE;   // I632.3
      "I632.4" { ExternalVisible := 'False'} : Bool := FALSE;   // I632.4
      "I632.5" { ExternalVisible := 'False'} : Bool := FALSE;   // I632.5
      "I632.6" { ExternalVisible := 'False'} : Bool := FALSE;   // I632.6
      "I632.7" { ExternalVisible := 'False'} : Bool := FALSE;   // I632.7
      "I633.0" { ExternalVisible := 'False'} : Bool := FALSE;   // I633.0
      "I633.1" { ExternalVisible := 'False'} : Bool := FALSE;   // I633.1
      "I633.2" { ExternalVisible := 'False'} : Bool := FALSE;   // I633.2
      "I633.3" { ExternalVisible := 'False'} : Bool := FALSE;   // I633.3
      "I633.4" { ExternalVisible := 'False'} : Bool := FALSE;   // I633.4
      "I633.5" { ExternalVisible := 'False'} : Bool := FALSE;   // I633.5
      "I633.6" { ExternalVisible := 'False'} : Bool := FALSE;   // I633.6
      "I633.7" { ExternalVisible := 'False'} : Bool := FALSE;   // I633.7
      "I634.0" { ExternalVisible := 'False'} : Bool := FALSE;   // I634.0
      "I634.1" { ExternalVisible := 'False'} : Bool := FALSE;   // I634.1
      "I634.2" { ExternalVisible := 'False'} : Bool := FALSE;   // I634.2
      "I634.3" { ExternalVisible := 'False'} : Bool := FALSE;   // I634.3
      "I634.4" { ExternalVisible := 'False'} : Bool := FALSE;   // I634.4
      "I634.5" { ExternalVisible := 'False'} : Bool := FALSE;   // I634.5
      "I634.6" { ExternalVisible := 'False'} : Bool := FALSE;   // I634.6
      "I634.7" { ExternalVisible := 'False'} : Bool := FALSE;   // I634.7
      "I635.0" { ExternalVisible := 'False'} : Bool := FALSE;   // I635.0
      "I635.1" { ExternalVisible := 'False'} : Bool := FALSE;   // I635.1
      "I635.2" { ExternalVisible := 'False'} : Bool := FALSE;   // I635.2
      "I635.3" { ExternalVisible := 'False'} : Bool := FALSE;   // I635.3
      "I635.4" { ExternalVisible := 'False'} : Bool := FALSE;   // I635.4
      "I635.5" { ExternalVisible := 'False'} : Bool := FALSE;   // I635.5
      "I635.6" { ExternalVisible := 'False'} : Bool := FALSE;   // I635.6
      "I635.7" { ExternalVisible := 'False'} : Bool := FALSE;   // I635.7
      "I636.0" { ExternalVisible := 'False'} : Bool := FALSE;   // I636.0
      "I636.1" { ExternalVisible := 'False'} : Bool := FALSE;   // I636.1
      "I636.2" { ExternalVisible := 'False'} : Bool := FALSE;   // I636.2
      "I636.3" { ExternalVisible := 'False'} : Bool := FALSE;   // I636.3
      "I636.4" { ExternalVisible := 'False'} : Bool := FALSE;   // I636.4
      "I636.5" { ExternalVisible := 'False'} : Bool := FALSE;   // I636.5
      "I636.6" { ExternalVisible := 'False'} : Bool := FALSE;   // I636.6
      "I636.7" { ExternalVisible := 'False'} : Bool := FALSE;   // I636.7
      "I637.0" { ExternalVisible := 'False'} : Bool := FALSE;   // I637.0
      "I637.1" { ExternalVisible := 'False'} : Bool := FALSE;   // I637.1
      "I637.2" { ExternalVisible := 'False'} : Bool := FALSE;   // I637.2
      "I637.3" { ExternalVisible := 'False'} : Bool := FALSE;   // I637.3
      "I637.4" { ExternalVisible := 'False'} : Bool := FALSE;   // I637.4
      "I637.5" { ExternalVisible := 'False'} : Bool := FALSE;   // I637.5
      "I637.6" { ExternalVisible := 'False'} : Bool := FALSE;   // I637.6
      "I637.7" { ExternalVisible := 'False'} : Bool := FALSE;   // I637.7
      "I638.0" { ExternalVisible := 'False'} : Bool := FALSE;   // I638.0
      "I638.1" { ExternalVisible := 'False'} : Bool := FALSE;   // I638.1
      "I638.2" { ExternalVisible := 'False'} : Bool := FALSE;   // I638.2
      "I638.3" { ExternalVisible := 'False'} : Bool := FALSE;   // I638.3
      "I638.4" { ExternalVisible := 'False'} : Bool := FALSE;   // I638.4
      "I638.5" { ExternalVisible := 'False'} : Bool := FALSE;   // I638.5
      "I638.6" { ExternalVisible := 'False'} : Bool := FALSE;   // I638.6
      "I638.7" { ExternalVisible := 'False'} : Bool := FALSE;   // I638.7
      "I639.0" { ExternalVisible := 'False'} : Bool := FALSE;   // I639.0
      "I639.1" { ExternalVisible := 'False'} : Bool := FALSE;   // I639.1
      "I639.2" { ExternalVisible := 'False'} : Bool := FALSE;   // I639.2
      "I639.3" { ExternalVisible := 'False'} : Bool := FALSE;   // I639.3
      "I639.4" { ExternalVisible := 'False'} : Bool := FALSE;   // I639.4
      "I639.5" { ExternalVisible := 'False'} : Bool := FALSE;   // I639.5
      "I639.6" { ExternalVisible := 'False'} : Bool := FALSE;   // I639.6
      "I639.7" { ExternalVisible := 'False'} : Bool := FALSE;   // I639.7
      "I640.0" { ExternalVisible := 'False'} : Bool := FALSE;   // I640.0
      "I640.1" { ExternalVisible := 'False'} : Bool := FALSE;   // I640.1
      "I640.2" { ExternalVisible := 'False'} : Bool := FALSE;   // I640.2
      "I640.3" { ExternalVisible := 'False'} : Bool := FALSE;   // I640.3
      "I640.4" { ExternalVisible := 'False'} : Bool := FALSE;   // I640.4
      "I640.5" { ExternalVisible := 'False'} : Bool := FALSE;   // I640.5
      "I640.6" { ExternalVisible := 'False'} : Bool := FALSE;   // I640.6
      "I640.7" { ExternalVisible := 'False'} : Bool := FALSE;   // I640.7
      "I641.0" { ExternalVisible := 'False'} : Bool := FALSE;   // I641.0
      "I641.1" { ExternalVisible := 'False'} : Bool := FALSE;   // I641.1
      "I641.2" { ExternalVisible := 'False'} : Bool := FALSE;   // I641.2
      "I641.3" { ExternalVisible := 'False'} : Bool := FALSE;   // I641.3
      "I641.4" { ExternalVisible := 'False'} : Bool := FALSE;   // I641.4
      "I641.5" { ExternalVisible := 'False'} : Bool := FALSE;   // I641.5
      "I641.6" { ExternalVisible := 'False'} : Bool := FALSE;   // I641.6
      "I641.7" { ExternalVisible := 'False'} : Bool := FALSE;   // I641.7
      "I642.0" { ExternalVisible := 'False'} : Bool := FALSE;   // I642.0
      "I642.1" { ExternalVisible := 'False'} : Bool := FALSE;   // I642.1
      "I642.2" { ExternalVisible := 'False'} : Bool := FALSE;   // I642.2
      "I642.3" { ExternalVisible := 'False'} : Bool := FALSE;   // I642.3
      "I642.4" { ExternalVisible := 'False'} : Bool := FALSE;   // I642.4
      "I642.5" { ExternalVisible := 'False'} : Bool := FALSE;   // I642.5
      "I642.6" { ExternalVisible := 'False'} : Bool := FALSE;   // I642.6
      "I642.7" { ExternalVisible := 'False'} : Bool := FALSE;   // I642.7
      "I643.0" { ExternalVisible := 'False'} : Bool := FALSE;   // I643.0
      "I643.1" { ExternalVisible := 'False'} : Bool := FALSE;   // I643.1
      "I643.2" { ExternalVisible := 'False'} : Bool := FALSE;   // I643.2
      "I643.3" { ExternalVisible := 'False'} : Bool := FALSE;   // I643.3
      "I643.4" { ExternalVisible := 'False'} : Bool := FALSE;   // I643.4
      "I643.5" { ExternalVisible := 'False'} : Bool := FALSE;   // I643.5
      "I643.6" { ExternalVisible := 'False'} : Bool := FALSE;   // I643.6
      "I643.7" { ExternalVisible := 'False'} : Bool := FALSE;   // I643.7
      "I644.0" { ExternalVisible := 'False'} : Bool := FALSE;   // I644.0
      "I644.1" { ExternalVisible := 'False'} : Bool := FALSE;   // I644.1
      "I644.2" { ExternalVisible := 'False'} : Bool := FALSE;   // I644.2
      "I644.3" { ExternalVisible := 'False'} : Bool := FALSE;   // I644.3
      "I644.4" { ExternalVisible := 'False'} : Bool := FALSE;   // I644.4
      "I644.5" { ExternalVisible := 'False'} : Bool := FALSE;   // I644.5
      "I644.6" { ExternalVisible := 'False'} : Bool := FALSE;   // I644.6
      "I644.7" { ExternalVisible := 'False'} : Bool := FALSE;   // I644.7
      "I645.0" { ExternalVisible := 'False'} : Bool := FALSE;   // I645.0
      "I645.1" { ExternalVisible := 'False'} : Bool := FALSE;   // I645.1
      "I645.2" { ExternalVisible := 'False'} : Bool := FALSE;   // I645.2
      "I645.3" { ExternalVisible := 'False'} : Bool := FALSE;   // I645.3
      "I645.4" { ExternalVisible := 'False'} : Bool := FALSE;   // I645.4
      "I645.5" { ExternalVisible := 'False'} : Bool := FALSE;   // I645.5
      "I645.6" { ExternalVisible := 'False'} : Bool := FALSE;   // I645.6
      "I645.7" { ExternalVisible := 'False'} : Bool := FALSE;   // I645.7
      "I646.0" { ExternalVisible := 'False'} : Bool := FALSE;   // I646.0
      "I646.1" { ExternalVisible := 'False'} : Bool := FALSE;   // I646.1
      "I646.2" { ExternalVisible := 'False'} : Bool := FALSE;   // I646.2
      "I646.3" { ExternalVisible := 'False'} : Bool := FALSE;   // I646.3
      "I646.4" { ExternalVisible := 'False'} : Bool := FALSE;   // I646.4
      "I646.5" { ExternalVisible := 'False'} : Bool := FALSE;   // I646.5
      "I646.6" { ExternalVisible := 'False'} : Bool := FALSE;   // I646.6
      "I646.7" { ExternalVisible := 'False'} : Bool := FALSE;   // I646.7
      "I647.0" { ExternalVisible := 'False'} : Bool := FALSE;   // I647.0
      "I647.1" { ExternalVisible := 'False'} : Bool := FALSE;   // I647.1
      "I647.2" { ExternalVisible := 'False'} : Bool := FALSE;   // I647.2
      "I647.3" { ExternalVisible := 'False'} : Bool := FALSE;   // I647.3
      "I647.4" { ExternalVisible := 'False'} : Bool := FALSE;   // I647.4
      "I647.5" { ExternalVisible := 'False'} : Bool := FALSE;   // I647.5
      "I647.6" { ExternalVisible := 'False'} : Bool := FALSE;   // I647.6
      "I647.7" { ExternalVisible := 'False'} : Bool := FALSE;   // I647.7
      "I648.0" { ExternalVisible := 'False'} : Bool := FALSE;   // I648.0
      "I648.1" { ExternalVisible := 'False'} : Bool := FALSE;   // I648.1
      "I648.2" { ExternalVisible := 'False'} : Bool := FALSE;   // I648.2
      "I648.3" { ExternalVisible := 'False'} : Bool := FALSE;   // I648.3
      "I648.4" { ExternalVisible := 'False'} : Bool := FALSE;   // I648.4
      "I648.5" { ExternalVisible := 'False'} : Bool := FALSE;   // I648.5
      "I648.6" { ExternalVisible := 'False'} : Bool := FALSE;   // I648.6
      "I648.7" { ExternalVisible := 'False'} : Bool := FALSE;   // I648.7
      "I649.0" { ExternalVisible := 'False'} : Bool := FALSE;   // I649.0
      "I649.1" { ExternalVisible := 'False'} : Bool := FALSE;   // I649.1
      "I649.2" { ExternalVisible := 'False'} : Bool := FALSE;   // I649.2
      "I649.3" { ExternalVisible := 'False'} : Bool := FALSE;   // I649.3
      "I649.4" { ExternalVisible := 'False'} : Bool := FALSE;   // I649.4
      "I649.5" { ExternalVisible := 'False'} : Bool := FALSE;   // I649.5
      "I649.6" { ExternalVisible := 'False'} : Bool := FALSE;   // I649.6
      "I649.7" { ExternalVisible := 'False'} : Bool := FALSE;   // I649.7
      "I650.0" { ExternalVisible := 'False'} : Bool := FALSE;   // I650.0
      "I650.1" { ExternalVisible := 'False'} : Bool := FALSE;   // I650.1
      "I650.2" { ExternalVisible := 'False'} : Bool := FALSE;   // I650.2
      "I650.3" { ExternalVisible := 'False'} : Bool := FALSE;   // I650.3
      "I650.4" { ExternalVisible := 'False'} : Bool := FALSE;   // I650.4
      "I650.5" { ExternalVisible := 'False'} : Bool := FALSE;   // I650.5
      "I650.6" { ExternalVisible := 'False'} : Bool := FALSE;   // I650.6
      "I650.7" { ExternalVisible := 'False'} : Bool := FALSE;   // I650.7
      "I651.0" { ExternalVisible := 'False'} : Bool := FALSE;   // I651.0
      "I651.1" { ExternalVisible := 'False'} : Bool := FALSE;   // I651.1
      "I651.2" { ExternalVisible := 'False'} : Bool := FALSE;   // I651.2
      "I651.3" { ExternalVisible := 'False'} : Bool := FALSE;   // I651.3
      "I651.4" { ExternalVisible := 'False'} : Bool := FALSE;   // I651.4
      "I651.5" { ExternalVisible := 'False'} : Bool := FALSE;   // I651.5
      "I651.6" { ExternalVisible := 'False'} : Bool := FALSE;   // I651.6
      "I651.7" { ExternalVisible := 'False'} : Bool := FALSE;   // I651.7
      "I652.0" { ExternalVisible := 'False'} : Bool := FALSE;   // I652.0
      "I652.1" { ExternalVisible := 'False'} : Bool := FALSE;   // I652.1
      "I652.2" { ExternalVisible := 'False'} : Bool := FALSE;   // I652.2
      "I652.3" { ExternalVisible := 'False'} : Bool := FALSE;   // I652.3
      "I652.4" { ExternalVisible := 'False'} : Bool := FALSE;   // I652.4
      "I652.5" { ExternalVisible := 'False'} : Bool := FALSE;   // I652.5
      "I652.6" { ExternalVisible := 'False'} : Bool := FALSE;   // I652.6
      "I652.7" { ExternalVisible := 'False'} : Bool := FALSE;   // I652.7
      "I653.0" { ExternalVisible := 'False'} : Bool := FALSE;   // I653.0
      "I653.1" { ExternalVisible := 'False'} : Bool := FALSE;   // I653.1
      "I653.2" { ExternalVisible := 'False'} : Bool := FALSE;   // I653.2
      "I653.3" { ExternalVisible := 'False'} : Bool := FALSE;   // I653.3
      "I653.4" { ExternalVisible := 'False'} : Bool := FALSE;   // I653.4
      "I653.5" { ExternalVisible := 'False'} : Bool := FALSE;   // I653.5
      "I653.6" { ExternalVisible := 'False'} : Bool := FALSE;   // I653.6
      "I653.7" { ExternalVisible := 'False'} : Bool := FALSE;   // I653.7
      "I654.0" { ExternalVisible := 'False'} : Bool := FALSE;   // I654.0
      "I654.1" { ExternalVisible := 'False'} : Bool := FALSE;   // I654.1
      "I654.2" { ExternalVisible := 'False'} : Bool := FALSE;   // I654.2
      "I654.3" { ExternalVisible := 'False'} : Bool := FALSE;   // I654.3
      "I654.4" { ExternalVisible := 'False'} : Bool := FALSE;   // I654.4
      "I654.5" { ExternalVisible := 'False'} : Bool := FALSE;   // I654.5
      "I654.6" { ExternalVisible := 'False'} : Bool := FALSE;   // I654.6
      "I654.7" { ExternalVisible := 'False'} : Bool := FALSE;   // I654.7
      "I655.0" { ExternalVisible := 'False'} : Bool := FALSE;   // I655.0
      "I655.1" { ExternalVisible := 'False'} : Bool := FALSE;   // I655.1
      "I655.2" { ExternalVisible := 'False'} : Bool := FALSE;   // I655.2
      "I655.3" { ExternalVisible := 'False'} : Bool := FALSE;   // I655.3
      "I655.4" { ExternalVisible := 'False'} : Bool := FALSE;   // I655.4
      "I655.5" { ExternalVisible := 'False'} : Bool := FALSE;   // I655.5
      "I655.6" { ExternalVisible := 'False'} : Bool := FALSE;   // I655.6
      "I655.7" { ExternalVisible := 'False'} : Bool := FALSE;   // I655.7
      "I656.0" { ExternalVisible := 'False'} : Bool := FALSE;   // I656.0
      "I656.1" { ExternalVisible := 'False'} : Bool := FALSE;   // I656.1
      "I656.2" { ExternalVisible := 'False'} : Bool := FALSE;   // I656.2
      "I656.3" { ExternalVisible := 'False'} : Bool := FALSE;   // I656.3
      "I656.4" { ExternalVisible := 'False'} : Bool := FALSE;   // I656.4
      "I656.5" { ExternalVisible := 'False'} : Bool := FALSE;   // I656.5
      "I656.6" { ExternalVisible := 'False'} : Bool := FALSE;   // I656.6
      "I656.7" { ExternalVisible := 'False'} : Bool := FALSE;   // I656.7
      "I657.0" { ExternalVisible := 'False'} : Bool := FALSE;   // I657.0
      "I657.1" { ExternalVisible := 'False'} : Bool := FALSE;   // I657.1
      "I657.2" { ExternalVisible := 'False'} : Bool := FALSE;   // I657.2
      "I657.3" { ExternalVisible := 'False'} : Bool := FALSE;   // I657.3
      "I657.4" { ExternalVisible := 'False'} : Bool := FALSE;   // I657.4
      "I657.5" { ExternalVisible := 'False'} : Bool := FALSE;   // I657.5
      "I657.6" { ExternalVisible := 'False'} : Bool := FALSE;   // I657.6
      "I657.7" { ExternalVisible := 'False'} : Bool := FALSE;   // I657.7
      "I658.0" { ExternalVisible := 'False'} : Bool := FALSE;   // I658.0
      "I658.1" { ExternalVisible := 'False'} : Bool := FALSE;   // I658.1
      "I658.2" { ExternalVisible := 'False'} : Bool := FALSE;   // I658.2
      "I658.3" { ExternalVisible := 'False'} : Bool := FALSE;   // I658.3
      "I658.4" { ExternalVisible := 'False'} : Bool := FALSE;   // I658.4
      "I658.5" { ExternalVisible := 'False'} : Bool := FALSE;   // I658.5
      "I658.6" { ExternalVisible := 'False'} : Bool := FALSE;   // I658.6
      "I658.7" { ExternalVisible := 'False'} : Bool := FALSE;   // I658.7
      "I659.0" { ExternalVisible := 'False'} : Bool := FALSE;   // I659.0
      "I659.1" { ExternalVisible := 'False'} : Bool := FALSE;   // I659.1
      "I659.2" { ExternalVisible := 'False'} : Bool := FALSE;   // I659.2
      "I659.3" { ExternalVisible := 'False'} : Bool := FALSE;   // I659.3
      "I659.4" { ExternalVisible := 'False'} : Bool := FALSE;   // I659.4
      "I659.5" { ExternalVisible := 'False'} : Bool := FALSE;   // I659.5
      "I659.6" { ExternalVisible := 'False'} : Bool := FALSE;   // I659.6
      "I659.7" { ExternalVisible := 'False'} : Bool := FALSE;   // I659.7
      "I660.0" { ExternalVisible := 'False'} : Bool := FALSE;   // I660.0
      "I660.1" { ExternalVisible := 'False'} : Bool := FALSE;   // I660.1
      "I660.2" { ExternalVisible := 'False'} : Bool := FALSE;   // I660.2
      "I660.3" { ExternalVisible := 'False'} : Bool := FALSE;   // I660.3
      "I660.4" { ExternalVisible := 'False'} : Bool := FALSE;   // I660.4
      "I660.5" { ExternalVisible := 'False'} : Bool := FALSE;   // I660.5
      "I660.6" { ExternalVisible := 'False'} : Bool := FALSE;   // I660.6
      "I660.7" { ExternalVisible := 'False'} : Bool := FALSE;   // I660.7
      "I661.0" { ExternalVisible := 'False'} : Bool := FALSE;   // I661.0
      "I661.1" { ExternalVisible := 'False'} : Bool := FALSE;   // I661.1
      "I661.2" { ExternalVisible := 'False'} : Bool := FALSE;   // I661.2
      "I661.3" { ExternalVisible := 'False'} : Bool := FALSE;   // I661.3
      "I661.4" { ExternalVisible := 'False'} : Bool := FALSE;   // I661.4
      "I661.5" { ExternalVisible := 'False'} : Bool := FALSE;   // I661.5
